REGION Network 6: Current revision and modification history
   // ▄▄▄▄▄▄▄▄▄▄▄▄▄▄▄▄▄▄▄▄▄▄▄▄▄▄▄▄▄▄▄▄▄▄▄▄▄▄▄▄▄▄▄▄
   // MODIFICATION HISTORY
   // 
   // 
   // The revision data shown here, in the network comments, contains additional information 
   // reflecting the software development workflow under the version control system (VCS) employed 
   // to track all software changes.
   // 
   // The VCS in use is the Git Source Code Management system in conjunction with the GitHub online 
   // hosting system. The software in its entirety is available in the GitHub remote repository:
   // 
   //      https://github.com/practicalseries/PS2001-pal-software
   // 
   // The repository is public and can be freely copied (forked in GitHub terminology) and used 
   // under the MIT licence. 
   // 
   // The MIT licence is reproduced in full in the last network of this software module.
   // 
   // 
   //  ―――――――――――――――――――――――――――――――――――――――――――
   //  DATE       REVISION             MASTER BRANCH     DEV
   //          (nnn.amm)   COMMIT TAG    (Base ---> Merge)    BRANCH   Author
   //  ———————————————————————————————————————————
   //  2022.04.16    002.000   D0011      D0010 D0011  None    M. Gledhill
   //                        FC11001 — RELEASED FOR USE
   //                          Merge back to master branch
   // 
   //  2022.04.11    001.801   D0010A-000.801   D0010 N/A     D010A   M. Gledhill
   //                        Released for test (SCV)
   // 
   //  2022.04.06    001.101   D0010A-000.104   D0010 N/A     D010A   M. Gledhill
   //                        Comments updated and standardised
   // 
   //  2021.08.23    001.000   D0009      D0008 D0009  None    M. Gledhill
   //                        FC11001 — RELEASED FOR USE
   //                          Merge back to master branch
   // 
   //  2021.08.23    001.000   D0008A-001.000   D0008 N/A     D0008A   M. Gledhill
   //                        FC11001 — Post-test RELEASED FOR USE
   // 
   //  2021.08.17    000.801   D0008A-000.801   D0008 N/A     D0008A   M. Gledhill
   //                        FC11001 Released for SMT
   // 
   //  2021.08.10    000.103   D0008A-000.103   D0008 N/A     D0008A   M. Gledhill
   //                        FC11001 Initial development testing
   // 
   //  2021.07.21    000.102   D0008A-000.102   D0008 N/A     D0008A   M. Gledhill
   //                        FC11001 Incremental build
   // 
   //  2021.07.13    000.101   D0008A-000.101   D0008 N/A     D0008A   M. Gledhill
   //                        FC11001 Block created — Comments added
   //  ———————————————————————————————————————————
   //   Where: nnn  =  Major revision
   //         a  =  Type (1-7 Development, 8 Proving, 9 Qualification, 0 Release)
   //       mm  =  Minor revision (must be 00 if a = 0)
   //         Block properties version number should be set to nn.a (only one decimal place)
   // 
   // ▄▄▄▄▄▄▄▄▄▄▄▄▄▄▄▄▄▄▄▄▄▄▄▄▄▄▄▄▄▄▄▄▄▄▄▄▄▄▄▄▄▄▄▄
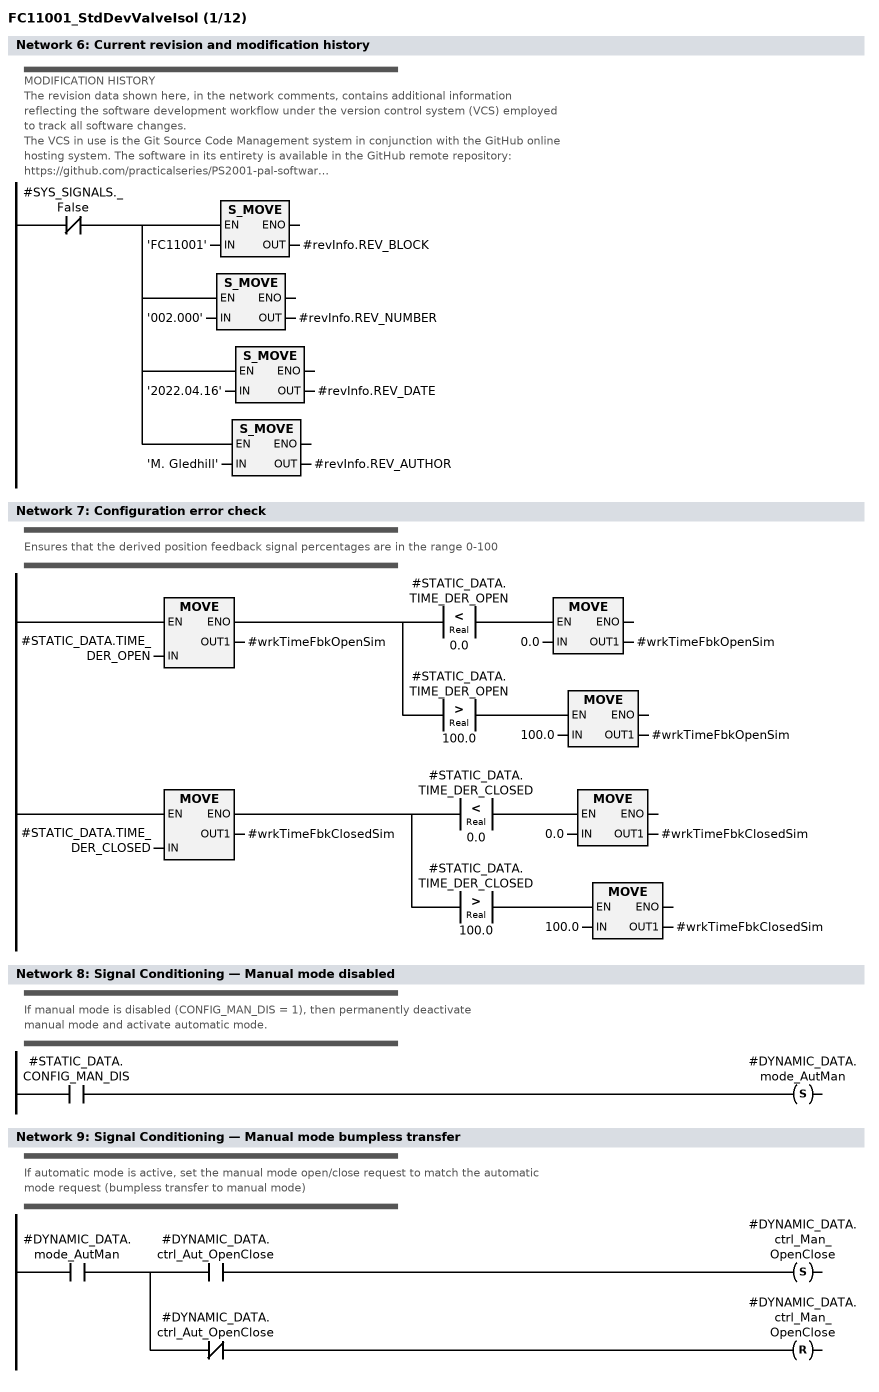
   RUNG wire#powerrail
      I_Contact( #SYS_SIGNALS._False )
      wire#w1
      S_Move(in := 'FC11001', out => #revInfo.REV_BLOCK)
   END_RUNG
   RUNG wire#w1
      S_Move(in := '002.000', out => #revInfo.REV_NUMBER)
   END_RUNG
   RUNG wire#w1
      S_Move(in := '2022.04.16', out => #revInfo.REV_DATE)
   END_RUNG
   RUNG wire#w1
      S_Move(in := 'M. Gledhill', out => #revInfo.REV_AUTHOR)
   END_RUNG
   // the same network as SCL:
   IF NOT #SYS_SIGNALS._False THEN
       #revInfo.REV_BLOCK := 'FC11001';
       #revInfo.REV_NUMBER := '002.000';
       #revInfo.REV_DATE := '2022.04.16';
       #revInfo.REV_AUTHOR := 'M. Gledhill';
   END_IF;
END_REGION

REGION Network 7: Configuration error check
   // ▀▀▀▀▀▀▀▀▀▀▀▀▀▀▀▀▀▀▀▀▀▀▀▀▀▀▀▀▀▀▀▀▀▀▀▀▀▀▀▀▀▀▀▀
   // Ensures that the derived position feedback signal percentages are in the range 0-100
   // ▄▄▄▄▄▄▄▄▄▄▄▄▄▄▄▄▄▄▄▄▄▄▄▄▄▄▄▄▄▄▄▄▄▄▄▄▄▄▄▄▄▄▄▄
   RUNG wire#powerrail
      Move(in := #STATIC_DATA.TIME_DER_OPEN, out1 => #wrkTimeFbkOpenSim)
      wire#w1
      { S7_Templates := "SrcType := Real" } LT_Contact(in1 := #STATIC_DATA.TIME_DER_OPEN, in2 := 0.0)
      Move(in := 0.0, out1 => #wrkTimeFbkOpenSim)
   END_RUNG
   RUNG wire#w1
      { S7_Templates := "SrcType := Real" } GT_Contact(in1 := #STATIC_DATA.TIME_DER_OPEN, in2 := 100.0)
      Move(in := 100.0, out1 => #wrkTimeFbkOpenSim)
   END_RUNG
   RUNG wire#powerrail
      Move(in := #STATIC_DATA.TIME_DER_CLOSED, out1 => #wrkTimeFbkClosedSim)
      wire#w2
      { S7_Templates := "SrcType := Real" } LT_Contact(in1 := #STATIC_DATA.TIME_DER_CLOSED, in2 := 0.0)
      Move(in := 0.0, out1 => #wrkTimeFbkClosedSim)
   END_RUNG
   RUNG wire#w2
      { S7_Templates := "SrcType := Real" } GT_Contact(in1 := #STATIC_DATA.TIME_DER_CLOSED, in2 := 100.0)
      Move(in := 100.0, out1 => #wrkTimeFbkClosedSim)
   END_RUNG
   // the same network as SCL:
   #wrkTimeFbkOpenSim := #STATIC_DATA.TIME_DER_OPEN;
   IF #STATIC_DATA.TIME_DER_OPEN < 0.0 THEN #wrkTimeFbkOpenSim := 0.0; END_IF;
   IF #STATIC_DATA.TIME_DER_OPEN > 100.0 THEN #wrkTimeFbkOpenSim := 100.0; END_IF;
   #wrkTimeFbkClosedSim := #STATIC_DATA.TIME_DER_CLOSED;
   IF #STATIC_DATA.TIME_DER_CLOSED < 0.0 THEN #wrkTimeFbkClosedSim := 0.0; END_IF;
   IF #STATIC_DATA.TIME_DER_CLOSED > 100.0 THEN #wrkTimeFbkClosedSim := 100.0; END_IF;
END_REGION

REGION Network 8: Signal Conditioning — Manual mode disabled
   // ▀▀▀▀▀▀▀▀▀▀▀▀▀▀▀▀▀▀▀▀▀▀▀▀▀▀▀▀▀▀▀▀▀▀▀▀▀▀▀▀▀▀▀▀
   // If manual mode is disabled (CONFIG_MAN_DIS = 1), then permanently deactivate
   // manual mode and activate automatic mode.
   // ▄▄▄▄▄▄▄▄▄▄▄▄▄▄▄▄▄▄▄▄▄▄▄▄▄▄▄▄▄▄▄▄▄▄▄▄▄▄▄▄▄▄▄▄
   RUNG wire#powerrail
      Contact( #STATIC_DATA.CONFIG_MAN_DIS )
      S_Coil( #DYNAMIC_DATA.mode_AutMan )
   END_RUNG
   // the same network as SCL:
   IF #STATIC_DATA.CONFIG_MAN_DIS THEN #DYNAMIC_DATA.mode_AutMan := TRUE; END_IF;
END_REGION

REGION Network 9: Signal Conditioning — Manual mode bumpless transfer
   // ▀▀▀▀▀▀▀▀▀▀▀▀▀▀▀▀▀▀▀▀▀▀▀▀▀▀▀▀▀▀▀▀▀▀▀▀▀▀▀▀▀▀▀▀
   // If automatic mode is active, set the manual mode open/close request to match the automatic
   // mode request (bumpless transfer to manual mode)
   // ▄▄▄▄▄▄▄▄▄▄▄▄▄▄▄▄▄▄▄▄▄▄▄▄▄▄▄▄▄▄▄▄▄▄▄▄▄▄▄▄▄▄▄▄
   RUNG wire#powerrail
      Contact( #DYNAMIC_DATA.mode_AutMan )
      wire#w1
      Contact( #DYNAMIC_DATA.ctrl_Aut_OpenClose )
      S_Coil( #DYNAMIC_DATA.ctrl_Man_OpenClose )
   END_RUNG
   RUNG wire#w1
      I_Contact( #DYNAMIC_DATA.ctrl_Aut_OpenClose )
      R_Coil( #DYNAMIC_DATA.ctrl_Man_OpenClose )
   END_RUNG
   // the same network as SCL:
   IF #DYNAMIC_DATA.mode_AutMan AND #DYNAMIC_DATA.ctrl_Aut_OpenClose THEN
       #DYNAMIC_DATA.ctrl_Man_OpenClose := TRUE;
   END_IF;
   IF #DYNAMIC_DATA.mode_AutMan AND NOT #DYNAMIC_DATA.ctrl_Aut_OpenClose THEN
       #DYNAMIC_DATA.ctrl_Man_OpenClose := FALSE;
   END_IF;
END_REGION

REGION Network 10: Signal Conditioning — Bypass mode disabled
   // ▀▀▀▀▀▀▀▀▀▀▀▀▀▀▀▀▀▀▀▀▀▀▀▀▀▀▀▀▀▀▀▀▀▀▀▀▀▀▀▀▀▀▀▀
   // If bypass mode is disabled (CONFIG_BYPASS_DIS = 1), then permanently deactivate
   // bypass mode.
   // ▄▄▄▄▄▄▄▄▄▄▄▄▄▄▄▄▄▄▄▄▄▄▄▄▄▄▄▄▄▄▄▄▄▄▄▄▄▄▄▄▄▄▄▄
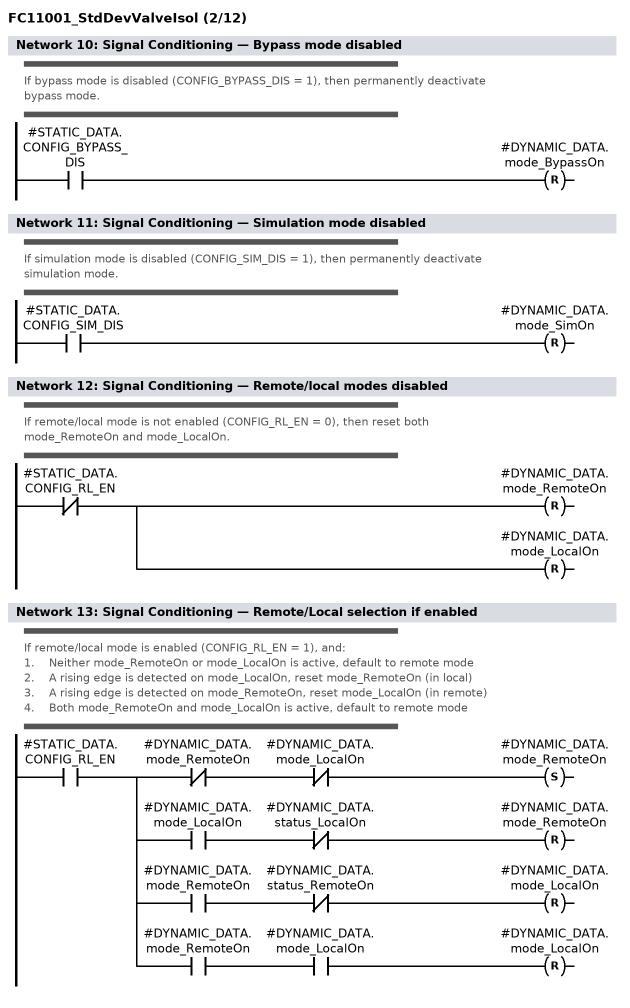
   RUNG wire#powerrail
      Contact( #STATIC_DATA.CONFIG_BYPASS_DIS )
      R_Coil( #DYNAMIC_DATA.mode_BypassOn )
   END_RUNG
   // the same network as SCL:
   IF #STATIC_DATA.CONFIG_BYPASS_DIS THEN #DYNAMIC_DATA.mode_BypassOn := FALSE; END_IF;
END_REGION

REGION Network 11: Signal Conditioning — Simulation mode disabled
   // ▀▀▀▀▀▀▀▀▀▀▀▀▀▀▀▀▀▀▀▀▀▀▀▀▀▀▀▀▀▀▀▀▀▀▀▀▀▀▀▀▀▀▀▀
   // If simulation mode is disabled (CONFIG_SIM_DIS = 1), then permanently deactivate
   // simulation mode.
   // ▄▄▄▄▄▄▄▄▄▄▄▄▄▄▄▄▄▄▄▄▄▄▄▄▄▄▄▄▄▄▄▄▄▄▄▄▄▄▄▄▄▄▄▄
   RUNG wire#powerrail
      Contact( #STATIC_DATA.CONFIG_SIM_DIS )
      R_Coil( #DYNAMIC_DATA.mode_SimOn )
   END_RUNG
   // the same network as SCL:
   IF #STATIC_DATA.CONFIG_SIM_DIS THEN #DYNAMIC_DATA.mode_SimOn := FALSE; END_IF;
END_REGION

REGION Network 12: Signal Conditioning — Remote/local modes disabled
   // ▀▀▀▀▀▀▀▀▀▀▀▀▀▀▀▀▀▀▀▀▀▀▀▀▀▀▀▀▀▀▀▀▀▀▀▀▀▀▀▀▀▀▀▀
   // If remote/local mode is not enabled (CONFIG_RL_EN = 0), then reset both 
   // mode_RemoteOn and mode_LocalOn.
   // ▄▄▄▄▄▄▄▄▄▄▄▄▄▄▄▄▄▄▄▄▄▄▄▄▄▄▄▄▄▄▄▄▄▄▄▄▄▄▄▄▄▄▄▄
   RUNG wire#powerrail
      I_Contact( #STATIC_DATA.CONFIG_RL_EN )
      wire#w1
      R_Coil( #DYNAMIC_DATA.mode_RemoteOn )
   END_RUNG
   RUNG wire#w1
      R_Coil( #DYNAMIC_DATA.mode_LocalOn )
   END_RUNG
   // the same network as SCL:
   IF NOT #STATIC_DATA.CONFIG_RL_EN THEN
       #DYNAMIC_DATA.mode_RemoteOn := FALSE;
       #DYNAMIC_DATA.mode_LocalOn := FALSE;
   END_IF;
END_REGION

REGION Network 13: Signal Conditioning — Remote/Local selection if enabled
   // ▀▀▀▀▀▀▀▀▀▀▀▀▀▀▀▀▀▀▀▀▀▀▀▀▀▀▀▀▀▀▀▀▀▀▀▀▀▀▀▀▀▀▀▀
   // If remote/local mode is enabled (CONFIG_RL_EN = 1), and:
   // 
   //    1.  Neither mode_RemoteOn or mode_LocalOn is active, default to remote mode
   //    2.  A rising edge is detected on mode_LocalOn, reset mode_RemoteOn (in local)
   //    3.  A rising edge is detected on mode_RemoteOn, reset mode_LocalOn (in remote)
   //    4.  Both mode_RemoteOn and mode_LocalOn is active, default to remote mode
   // ▄▄▄▄▄▄▄▄▄▄▄▄▄▄▄▄▄▄▄▄▄▄▄▄▄▄▄▄▄▄▄▄▄▄▄▄▄▄▄▄▄▄▄▄
   RUNG wire#powerrail
      Contact( #STATIC_DATA.CONFIG_RL_EN )
      wire#w1
      I_Contact( #DYNAMIC_DATA.mode_RemoteOn )
      I_Contact( #DYNAMIC_DATA.mode_LocalOn )
      S_Coil( #DYNAMIC_DATA.mode_RemoteOn )
   END_RUNG
   RUNG wire#w1
      Contact( #DYNAMIC_DATA.mode_LocalOn )
      I_Contact( #DYNAMIC_DATA.status_LocalOn )
      R_Coil( #DYNAMIC_DATA.mode_RemoteOn )
   END_RUNG
   RUNG wire#w1
      Contact( #DYNAMIC_DATA.mode_RemoteOn )
      I_Contact( #DYNAMIC_DATA.status_RemoteOn )
      R_Coil( #DYNAMIC_DATA.mode_LocalOn )
   END_RUNG
   RUNG wire#w1
      Contact( #DYNAMIC_DATA.mode_RemoteOn )
      Contact( #DYNAMIC_DATA.mode_LocalOn )
      R_Coil( #DYNAMIC_DATA.mode_LocalOn )
   END_RUNG
   // the same network as SCL:
   IF #STATIC_DATA.CONFIG_RL_EN AND NOT #DYNAMIC_DATA.mode_RemoteOn AND NOT #DYNAMIC_DATA.mode_LocalOn THEN
       #DYNAMIC_DATA.mode_RemoteOn := TRUE;
   END_IF;
   IF #STATIC_DATA.CONFIG_RL_EN AND #DYNAMIC_DATA.mode_LocalOn AND NOT #DYNAMIC_DATA.status_LocalOn THEN
       #DYNAMIC_DATA.mode_RemoteOn := FALSE;
   END_IF;
   IF #STATIC_DATA.CONFIG_RL_EN AND #DYNAMIC_DATA.mode_RemoteOn AND NOT #DYNAMIC_DATA.status_RemoteOn THEN
       #DYNAMIC_DATA.mode_LocalOn := FALSE;
   END_IF;
   IF #STATIC_DATA.CONFIG_RL_EN AND #DYNAMIC_DATA.mode_RemoteOn AND #DYNAMIC_DATA.mode_LocalOn THEN
       #DYNAMIC_DATA.mode_LocalOn := FALSE;
   END_IF;
END_REGION

REGION Network 14: Signal Conditioning — Derived open position
   // ▀▀▀▀▀▀▀▀▀▀▀▀▀▀▀▀▀▀▀▀▀▀▀▀▀▀▀▀▀▀▀▀▀▀▀▀▀▀▀▀▀▀▀▀
   // If there is no open position feedback (CONFIG_FBK_OPEN_EN = 0), then the open state of the 
   // valve is derived from the elapsed time of the operation timer using the following formulae:
   // 
   // ┌───────────────────────────────────────────┐
   // │$derived_fbk_open =1 when:                                │
   // │                                 wrkTimeFbkOpenSim  │
   // │actual_Operating_Timer ≤ TIME_OPENING_MAX ─ TIME_OPENING_MAX ╳ ----------------------------------------│
   // │                                     100     │
   // └───────────────────────────────────────────┘
   // Note:    wrkTimeFbkOpenSim is the error checked equivalent of TIME_FBK_OPEN
   // 
   // If the calculated elapsed time is close to or less than k_TIME_OP_MIN (210ms),
   // the calculated elapsed time (calOpenElapsedTime) is set to k_TIME_OP_MIN. This ensures at
   // least one timing pulse is required before the timer reaches zero.
   // 
   // The derived open signal ($derived_fbk_open) is reset if the valve is requested to be closed
   // ($ctrl_OpenClose = 0).
   // ▄▄▄▄▄▄▄▄▄▄▄▄▄▄▄▄▄▄▄▄▄▄▄▄▄▄▄▄▄▄▄▄▄▄▄▄▄▄▄▄▄▄▄▄
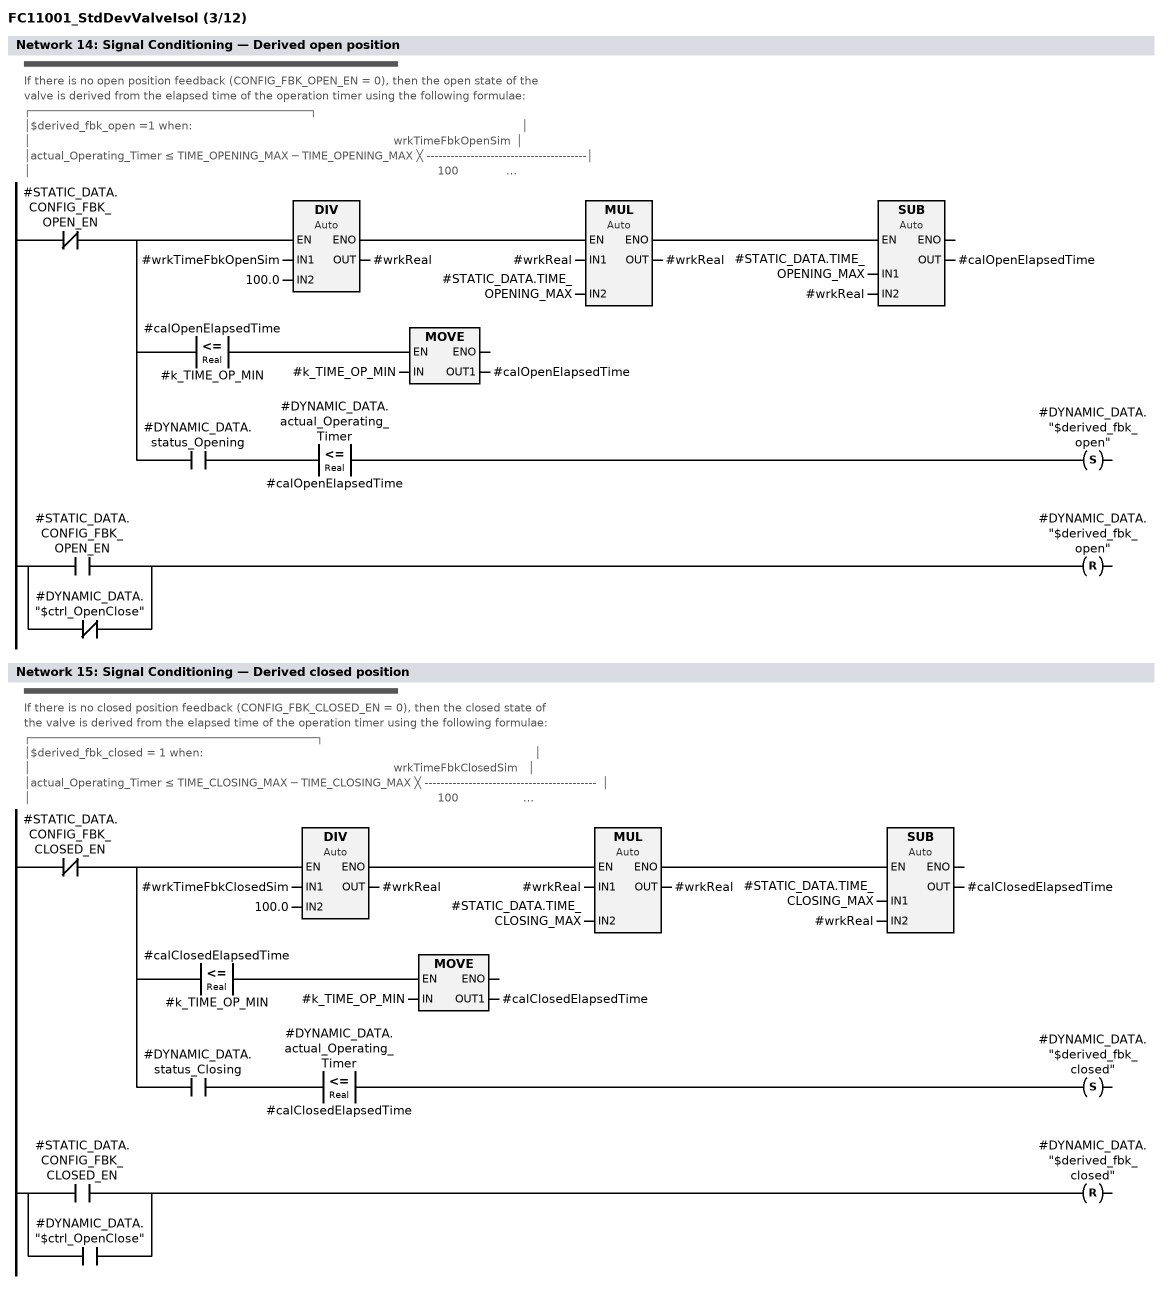
   RUNG wire#powerrail
      I_Contact( #STATIC_DATA.CONFIG_FBK_OPEN_EN )
      wire#w1
      Div(in1 := #wrkTimeFbkOpenSim, in2 := 100.0, out => #wrkReal)
      Mul(in1 := #wrkReal, in2 := #STATIC_DATA.TIME_OPENING_MAX, out => #wrkReal)
      Sub(in1 := #STATIC_DATA.TIME_OPENING_MAX, in2 := #wrkReal, out => #calOpenElapsedTime)
   END_RUNG
   RUNG wire#w1
      { S7_Templates := "SrcType := Real" } LE_Contact(in1 := #calOpenElapsedTime, in2 := #k_TIME_OP_MIN)
      Move(in := #k_TIME_OP_MIN, out1 => #calOpenElapsedTime)
   END_RUNG
   RUNG wire#w1
      Contact( #DYNAMIC_DATA.status_Opening )
      { S7_Templates := "SrcType := Real" } LE_Contact(in1 := #DYNAMIC_DATA.actual_Operating_Timer, in2 := #calOpenElapsedTime)
      S_Coil( #DYNAMIC_DATA."$derived_fbk_open" )
   END_RUNG
   RUNG wire#powerrail
      Contact( #STATIC_DATA.CONFIG_FBK_OPEN_EN )
      wire#w2
      R_Coil( #DYNAMIC_DATA."$derived_fbk_open" )
   END_RUNG
   RUNG wire#powerrail
      I_Contact( #DYNAMIC_DATA."$ctrl_OpenClose" )
   END_RUNG wire#w2
   // the same network as SCL:
   #_w1 := NOT #STATIC_DATA.CONFIG_FBK_OPEN_EN;
   IF #_w1 THEN
       #wrkReal := #wrkTimeFbkOpenSim / 100.0;
       #wrkReal := #wrkReal * #STATIC_DATA.TIME_OPENING_MAX;
       #calOpenElapsedTime := #STATIC_DATA.TIME_OPENING_MAX - #wrkReal;
   END_IF;
   IF #_w1 AND (#calOpenElapsedTime <= #k_TIME_OP_MIN) THEN #calOpenElapsedTime := #k_TIME_OP_MIN; END_IF;
   IF #_w1 AND #DYNAMIC_DATA.status_Opening AND (#DYNAMIC_DATA.actual_Operating_Timer <= #calOpenElapsedTime) THEN
       #DYNAMIC_DATA."$derived_fbk_open" := TRUE;
   END_IF;
   IF #STATIC_DATA.CONFIG_FBK_OPEN_EN OR NOT #DYNAMIC_DATA."$ctrl_OpenClose" THEN
       #DYNAMIC_DATA."$derived_fbk_open" := FALSE;
   END_IF;
END_REGION

REGION Network 15: Signal Conditioning — Derived closed position
   // ▀▀▀▀▀▀▀▀▀▀▀▀▀▀▀▀▀▀▀▀▀▀▀▀▀▀▀▀▀▀▀▀▀▀▀▀▀▀▀▀▀▀▀▀
   // If there is no closed position feedback (CONFIG_FBK_CLOSED_EN = 0), then the closed state of 
   // the valve is derived from the elapsed time of the operation timer using the following formulae:
   // 
   // ┌────────────────────────────────────────────┐
   // │$derived_fbk_closed = 1 when:                                 │
   // │                                 wrkTimeFbkClosedSim   │
   // │actual_Operating_Timer ≤ TIME_CLOSING_MAX ─ TIME_CLOSING_MAX ╳ -------------------------------------------  │
   // │                                     100            │
   // └────────────────────────────────────────────┘
   // Note:    wrkTimeFbkClosedSim is the error checked equivalent of TIME_FBK_CLOSED
   // 
   // If the calculated elapsed time is close to or less than k_TIME_OP_MIN (210ms),
   // the calculated elapsed time (calClosedElapsedTime) is set to k_TIME_OP_MIN. This ensures at
   // least one timing pulse is required before the timer reaches zero.
   // 
   // The derived closed signal ($derived_fbk_closed) is reset if the valve is requested to be open
   // ($ctrl_OpenClose = 1).
   // ▄▄▄▄▄▄▄▄▄▄▄▄▄▄▄▄▄▄▄▄▄▄▄▄▄▄▄▄▄▄▄▄▄▄▄▄▄▄▄▄▄▄▄▄
   RUNG wire#powerrail
      I_Contact( #STATIC_DATA.CONFIG_FBK_CLOSED_EN )
      wire#w1
      Div(in1 := #wrkTimeFbkClosedSim, in2 := 100.0, out => #wrkReal)
      Mul(in1 := #wrkReal, in2 := #STATIC_DATA.TIME_CLOSING_MAX, out => #wrkReal)
      Sub(in1 := #STATIC_DATA.TIME_CLOSING_MAX, in2 := #wrkReal, out => #calClosedElapsedTime)
   END_RUNG
   RUNG wire#w1
      { S7_Templates := "SrcType := Real" } LE_Contact(in1 := #calClosedElapsedTime, in2 := #k_TIME_OP_MIN)
      Move(in := #k_TIME_OP_MIN, out1 => #calClosedElapsedTime)
   END_RUNG
   RUNG wire#w1
      Contact( #DYNAMIC_DATA.status_Closing )
      { S7_Templates := "SrcType := Real" } LE_Contact(in1 := #DYNAMIC_DATA.actual_Operating_Timer, in2 := #calClosedElapsedTime)
      S_Coil( #DYNAMIC_DATA."$derived_fbk_closed" )
   END_RUNG
   RUNG wire#powerrail
      Contact( #STATIC_DATA.CONFIG_FBK_CLOSED_EN )
      wire#w2
      R_Coil( #DYNAMIC_DATA."$derived_fbk_closed" )
   END_RUNG
   RUNG wire#powerrail
      Contact( #DYNAMIC_DATA."$ctrl_OpenClose" )
   END_RUNG wire#w2
   // the same network as SCL:
   #_w1 := NOT #STATIC_DATA.CONFIG_FBK_CLOSED_EN;
   IF #_w1 THEN
       #wrkReal := #wrkTimeFbkClosedSim / 100.0;
       #wrkReal := #wrkReal * #STATIC_DATA.TIME_CLOSING_MAX;
       #calClosedElapsedTime := #STATIC_DATA.TIME_CLOSING_MAX - #wrkReal;
   END_IF;
   IF #_w1 AND (#calClosedElapsedTime <= #k_TIME_OP_MIN) THEN
       #calClosedElapsedTime := #k_TIME_OP_MIN;
   END_IF;
   IF #_w1 AND #DYNAMIC_DATA.status_Closing AND (#DYNAMIC_DATA.actual_Operating_Timer <= #calClosedElapsedTime) THEN
       #DYNAMIC_DATA."$derived_fbk_closed" := TRUE;
   END_IF;
   IF #STATIC_DATA.CONFIG_FBK_CLOSED_EN OR #DYNAMIC_DATA."$ctrl_OpenClose" THEN
       #DYNAMIC_DATA."$derived_fbk_closed" := FALSE;
   END_IF;
END_REGION

REGION Network 16: Signal Conditioning — Simulation mode — Open signal
   // ▀▀▀▀▀▀▀▀▀▀▀▀▀▀▀▀▀▀▀▀▀▀▀▀▀▀▀▀▀▀▀▀▀▀▀▀▀▀▀▀▀▀▀▀
   // If simulation mode is active, the simulated open position signal is set as follows:
   // 
   //    •   mode_SimValue = 0 (no feedback), $sim_fbk_open = 0
   // 
   //    •   mode_SimValue = 1 (permanently open), $sim_fbk_open = 1
   // 
   //    •   mode_SimValue = 2 (permanently closed), $sim_fbk_open = 0
   // 
   //    •   mode_SimValue = 3 (follow demand), $sim_fbk_open = $ctrl_OpenClose
   // 
   // If simulation mode is not active,  $sim_fbk_open = 0
   // ▄▄▄▄▄▄▄▄▄▄▄▄▄▄▄▄▄▄▄▄▄▄▄▄▄▄▄▄▄▄▄▄▄▄▄▄▄▄▄▄▄▄▄▄
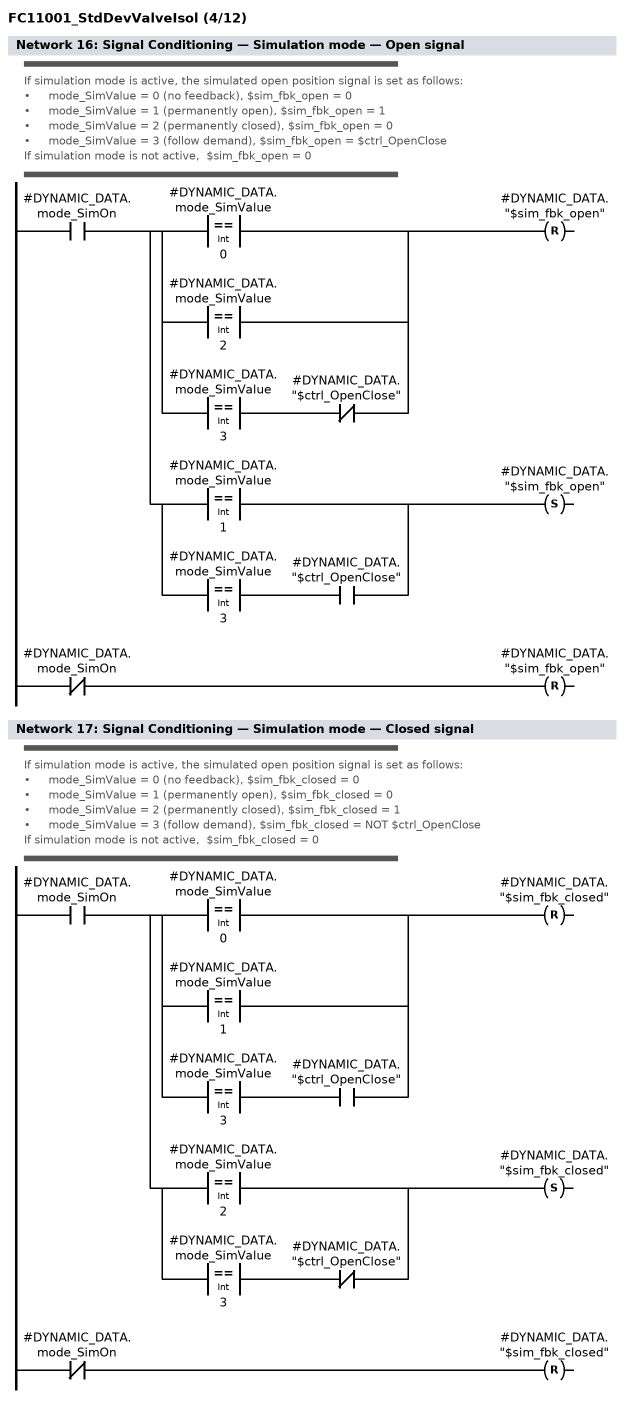
   RUNG wire#powerrail
      Contact( #DYNAMIC_DATA.mode_SimOn )
      wire#w1
      { S7_Templates := "SrcType := Int" } EQ_Contact(in1 := #DYNAMIC_DATA.mode_SimValue, in2 := 0)
      wire#w2
      R_Coil( #DYNAMIC_DATA."$sim_fbk_open" )
   END_RUNG
   RUNG wire#w1
      { S7_Templates := "SrcType := Int" } EQ_Contact(in1 := #DYNAMIC_DATA.mode_SimValue, in2 := 2)
   END_RUNG wire#w2
   RUNG wire#w1
      { S7_Templates := "SrcType := Int" } EQ_Contact(in1 := #DYNAMIC_DATA.mode_SimValue, in2 := 3)
      I_Contact( #DYNAMIC_DATA."$ctrl_OpenClose" )
   END_RUNG wire#w2
   RUNG wire#w1
      { S7_Templates := "SrcType := Int" } EQ_Contact(in1 := #DYNAMIC_DATA.mode_SimValue, in2 := 1)
      wire#w3
      S_Coil( #DYNAMIC_DATA."$sim_fbk_open" )
   END_RUNG
   RUNG wire#w1
      { S7_Templates := "SrcType := Int" } EQ_Contact(in1 := #DYNAMIC_DATA.mode_SimValue, in2 := 3)
      Contact( #DYNAMIC_DATA."$ctrl_OpenClose" )
   END_RUNG wire#w3
   RUNG wire#powerrail
      I_Contact( #DYNAMIC_DATA.mode_SimOn )
      R_Coil( #DYNAMIC_DATA."$sim_fbk_open" )
   END_RUNG
   // the same network as SCL:
   IF #DYNAMIC_DATA.mode_SimOn AND ((#DYNAMIC_DATA.mode_SimValue = 0) OR (#DYNAMIC_DATA.mode_SimValue = 2) OR ((#DYNAMIC_DATA.mode_SimValue = 3) AND NOT #DYNAMIC_DATA."$ctrl_OpenClose")) THEN
       #DYNAMIC_DATA."$sim_fbk_open" := FALSE;
   END_IF;
   IF #DYNAMIC_DATA.mode_SimOn AND ((#DYNAMIC_DATA.mode_SimValue = 1) OR ((#DYNAMIC_DATA.mode_SimValue = 3) AND #DYNAMIC_DATA."$ctrl_OpenClose")) THEN
       #DYNAMIC_DATA."$sim_fbk_open" := TRUE;
   END_IF;
   IF NOT #DYNAMIC_DATA.mode_SimOn THEN #DYNAMIC_DATA."$sim_fbk_open" := FALSE; END_IF;
END_REGION

REGION Network 17: Signal Conditioning — Simulation mode — Closed signal
   // ▀▀▀▀▀▀▀▀▀▀▀▀▀▀▀▀▀▀▀▀▀▀▀▀▀▀▀▀▀▀▀▀▀▀▀▀▀▀▀▀▀▀▀▀
   // If simulation mode is active, the simulated open position signal is set as follows:
   // 
   //    •   mode_SimValue = 0 (no feedback), $sim_fbk_closed = 0
   // 
   //    •   mode_SimValue = 1 (permanently open), $sim_fbk_closed = 0
   // 
   //    •   mode_SimValue = 2 (permanently closed), $sim_fbk_closed = 1
   // 
   //    •   mode_SimValue = 3 (follow demand), $sim_fbk_closed = NOT $ctrl_OpenClose
   // 
   // If simulation mode is not active,  $sim_fbk_closed = 0
   // ▄▄▄▄▄▄▄▄▄▄▄▄▄▄▄▄▄▄▄▄▄▄▄▄▄▄▄▄▄▄▄▄▄▄▄▄▄▄▄▄▄▄▄▄
   RUNG wire#powerrail
      Contact( #DYNAMIC_DATA.mode_SimOn )
      wire#w1
      { S7_Templates := "SrcType := Int" } EQ_Contact(in1 := #DYNAMIC_DATA.mode_SimValue, in2 := 0)
      wire#w2
      R_Coil( #DYNAMIC_DATA."$sim_fbk_closed" )
   END_RUNG
   RUNG wire#w1
      { S7_Templates := "SrcType := Int" } EQ_Contact(in1 := #DYNAMIC_DATA.mode_SimValue, in2 := 1)
   END_RUNG wire#w2
   RUNG wire#w1
      { S7_Templates := "SrcType := Int" } EQ_Contact(in1 := #DYNAMIC_DATA.mode_SimValue, in2 := 3)
      Contact( #DYNAMIC_DATA."$ctrl_OpenClose" )
   END_RUNG wire#w2
   RUNG wire#w1
      { S7_Templates := "SrcType := Int" } EQ_Contact(in1 := #DYNAMIC_DATA.mode_SimValue, in2 := 2)
      wire#w3
      S_Coil( #DYNAMIC_DATA."$sim_fbk_closed" )
   END_RUNG
   RUNG wire#w1
      { S7_Templates := "SrcType := Int" } EQ_Contact(in1 := #DYNAMIC_DATA.mode_SimValue, in2 := 3)
      I_Contact( #DYNAMIC_DATA."$ctrl_OpenClose" )
   END_RUNG wire#w3
   RUNG wire#powerrail
      I_Contact( #DYNAMIC_DATA.mode_SimOn )
      R_Coil( #DYNAMIC_DATA."$sim_fbk_closed" )
   END_RUNG
   // the same network as SCL:
   IF #DYNAMIC_DATA.mode_SimOn AND ((#DYNAMIC_DATA.mode_SimValue = 0) OR (#DYNAMIC_DATA.mode_SimValue = 1) OR ((#DYNAMIC_DATA.mode_SimValue = 3) AND #DYNAMIC_DATA."$ctrl_OpenClose")) THEN
       #DYNAMIC_DATA."$sim_fbk_closed" := FALSE;
   END_IF;
   IF #DYNAMIC_DATA.mode_SimOn AND ((#DYNAMIC_DATA.mode_SimValue = 2) OR ((#DYNAMIC_DATA.mode_SimValue = 3) AND NOT #DYNAMIC_DATA."$ctrl_OpenClose")) THEN
       #DYNAMIC_DATA."$sim_fbk_closed" := TRUE;
   END_IF;
   IF NOT #DYNAMIC_DATA.mode_SimOn THEN #DYNAMIC_DATA."$sim_fbk_closed" := FALSE; END_IF;
END_REGION

REGION Network 18: Signal conditioning — Determine valve OPEN position status
   // ▀▀▀▀▀▀▀▀▀▀▀▀▀▀▀▀▀▀▀▀▀▀▀▀▀▀▀▀▀▀▀▀▀▀▀▀▀▀▀▀▀▀▀▀
   // Generates a working open signal (wrkOpen), that is then used throughout the module as the 
   // definitive open position feedback signal.
   // 
   // The open signal will be either :
   // 
   //    1.  The same as the FBK_OPEN parameter if this is in use 
   //      (CONFIG_FBK_OPEN_EN = 1)
   // 
   //    2.  The internally derived open state (based on the requested state of the valve) if the 
   //      FBK_OPEN signal is NOT in use (CONFIG_FBK_OPEN_EN = 0)
   // 
   //    3.  The simulated state of the valve if simulation mode is active (mode_SimOn = 1)
   // 
   // If an actual open position signal is provided to the module via the FBK_OPEN parameter 
   // (i.e. if CONFIG_FBK_OPEN_EN = 1) then wrkOpen is set to match the FBK_OPEN signal 
   // (wrkOpen = FBK_OPEN).
   // 
   // If a derived open signal is to be used (i.e. if CONFIG_FBK_OPEN_EN = 0), then wrkOpen is set to 
   // match the internally derived $derived_fbk_open signal (wrkOpen = $derived_fbk_open). 
   // $derived_fbk_open is based on the requested state of the valve. 
   // 
   // Finally, if simulation mode is active (mode_SimOn = 1), then wrkOpen is set to match the internal 
   // simulation signal $sim_fbk_open signal (wrkOpen = $sim_fbk_open).. 
   // ▄▄▄▄▄▄▄▄▄▄▄▄▄▄▄▄▄▄▄▄▄▄▄▄▄▄▄▄▄▄▄▄▄▄▄▄▄▄▄▄▄▄▄▄
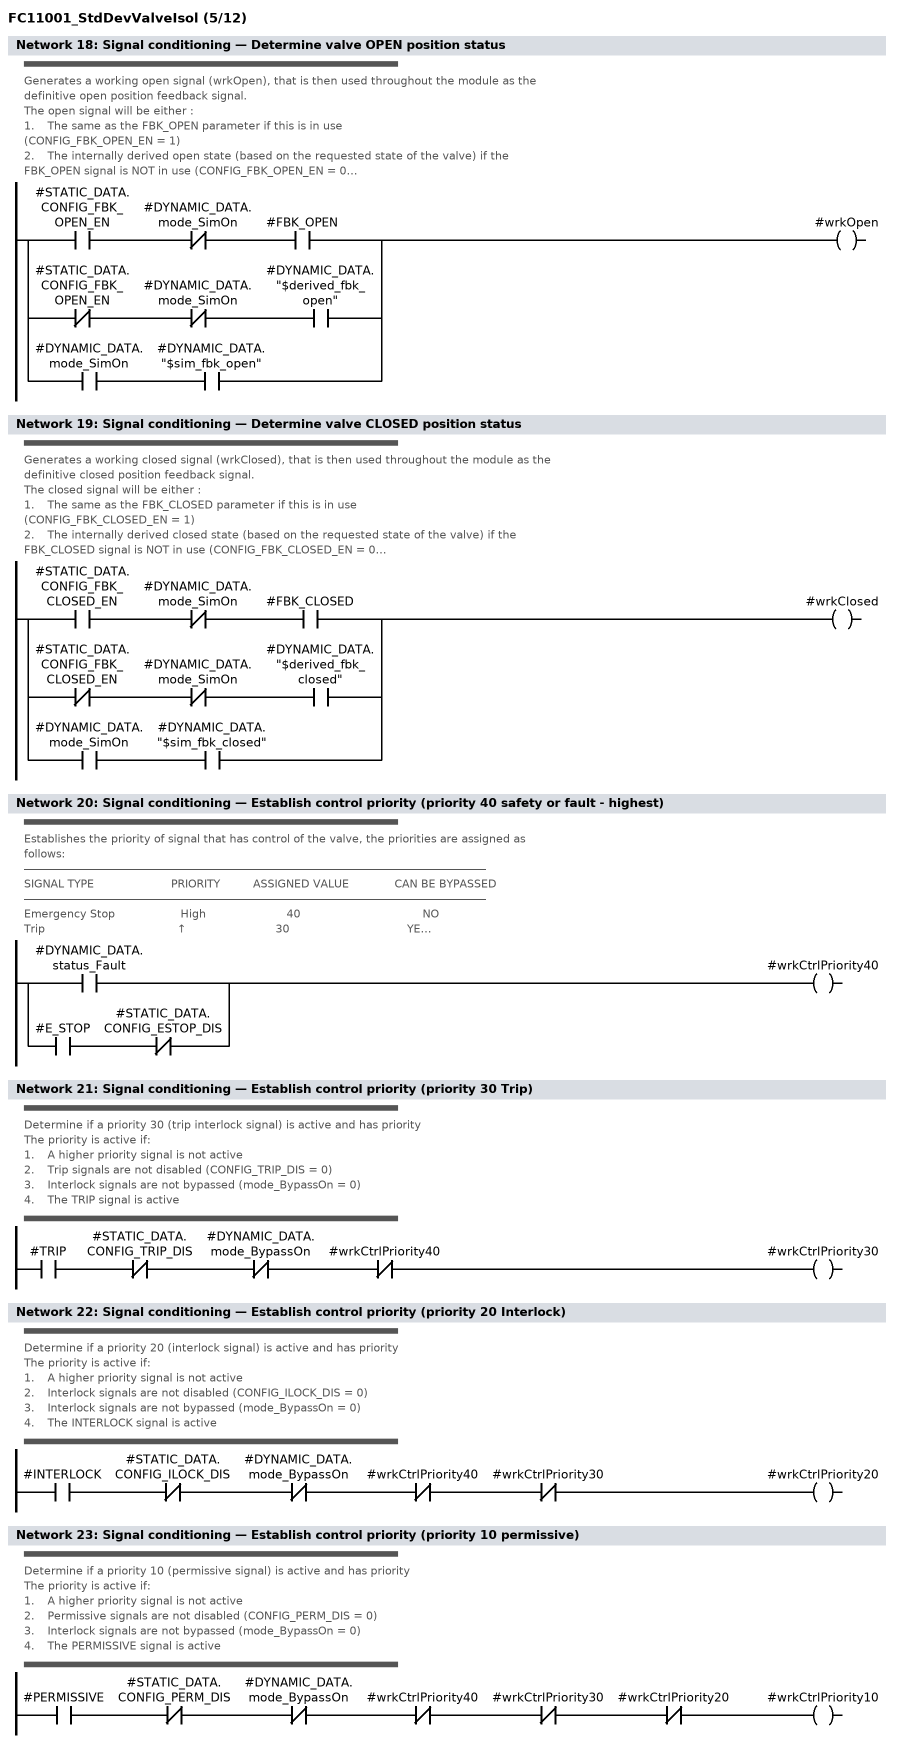
   RUNG wire#powerrail
      Contact( #STATIC_DATA.CONFIG_FBK_OPEN_EN )
      I_Contact( #DYNAMIC_DATA.mode_SimOn )
      Contact( #FBK_OPEN )
      wire#w1
      Coil( #wrkOpen )
   END_RUNG
   RUNG wire#powerrail
      I_Contact( #STATIC_DATA.CONFIG_FBK_OPEN_EN )
      I_Contact( #DYNAMIC_DATA.mode_SimOn )
      Contact( #DYNAMIC_DATA."$derived_fbk_open" )
   END_RUNG wire#w1
   RUNG wire#powerrail
      Contact( #DYNAMIC_DATA.mode_SimOn )
      Contact( #DYNAMIC_DATA."$sim_fbk_open" )
   END_RUNG wire#w1
   // the same network as SCL:
   #wrkOpen := (#STATIC_DATA.CONFIG_FBK_OPEN_EN AND NOT #DYNAMIC_DATA.mode_SimOn AND #FBK_OPEN) OR (NOT #STATIC_DATA.CONFIG_FBK_OPEN_EN AND NOT #DYNAMIC_DATA.mode_SimOn AND #DYNAMIC_DATA."$derived_fbk_open") OR (#DYNAMIC_DATA.mode_SimOn AND #DYNAMIC_DATA."$sim_fbk_open");
END_REGION

REGION Network 19: Signal conditioning — Determine valve CLOSED position status
   // ▀▀▀▀▀▀▀▀▀▀▀▀▀▀▀▀▀▀▀▀▀▀▀▀▀▀▀▀▀▀▀▀▀▀▀▀▀▀▀▀▀▀▀▀
   // Generates a working closed signal (wrkClosed), that is then used throughout the module as the 
   // definitive closed position feedback signal.
   // 
   // The closed signal will be either :
   // 
   //    1.  The same as the FBK_CLOSED parameter if this is in use 
   //      (CONFIG_FBK_CLOSED_EN = 1)
   // 
   //    2.  The internally derived closed state (based on the requested state of the valve) if the 
   //      FBK_CLOSED signal is NOT in use (CONFIG_FBK_CLOSED_EN = 0)
   // 
   //    3.  The simulated state of the valve if simulation mode is active (mode_SimOn = 1)
   // 
   // If an actual closed position signal is provided to the module via the FBK_CLOSED parameter 
   // (i.e. if CONFIG_FBK_CLOSED_EN = 1) then wrkClosed is set to match the FBK_CLOSED signal 
   // wrkClosed = FBK_CLOSED).
   // 
   // If a derived closed signal is to be used (i.e. if CONFIG_FBK_CLOSED_EN = 0), then wrkClosed is 
   // set to match the internally derived $derived_fbk_closed signal 
   // (wrkClosed = $derived_fbk_closed). $derived_fbk_closed is based on the requested state of 
   // the valve.
   // 
   // Finally, if simulation mode is active (mode_SimOn = 1), then wrkClosed is set to match the 
   // internal simulation signal $sim_fbk_closed signal (wrkClosed = $sim_fbk_closed). 
   // ▄▄▄▄▄▄▄▄▄▄▄▄▄▄▄▄▄▄▄▄▄▄▄▄▄▄▄▄▄▄▄▄▄▄▄▄▄▄▄▄▄▄▄▄
   RUNG wire#powerrail
      Contact( #STATIC_DATA.CONFIG_FBK_CLOSED_EN )
      I_Contact( #DYNAMIC_DATA.mode_SimOn )
      Contact( #FBK_CLOSED )
      wire#w1
      Coil( #wrkClosed )
   END_RUNG
   RUNG wire#powerrail
      I_Contact( #STATIC_DATA.CONFIG_FBK_CLOSED_EN )
      I_Contact( #DYNAMIC_DATA.mode_SimOn )
      Contact( #DYNAMIC_DATA."$derived_fbk_closed" )
   END_RUNG wire#w1
   RUNG wire#powerrail
      Contact( #DYNAMIC_DATA.mode_SimOn )
      Contact( #DYNAMIC_DATA."$sim_fbk_closed" )
   END_RUNG wire#w1
   // the same network as SCL:
   #wrkClosed := (#STATIC_DATA.CONFIG_FBK_CLOSED_EN AND NOT #DYNAMIC_DATA.mode_SimOn AND #FBK_CLOSED) OR (NOT #STATIC_DATA.CONFIG_FBK_CLOSED_EN AND NOT #DYNAMIC_DATA.mode_SimOn AND #DYNAMIC_DATA."$derived_fbk_closed") OR (#DYNAMIC_DATA.mode_SimOn AND #DYNAMIC_DATA."$sim_fbk_closed");
END_REGION

REGION Network 20: Signal conditioning — Establish control priority (priority 40 safety or fault - highest)
   // ▀▀▀▀▀▀▀▀▀▀▀▀▀▀▀▀▀▀▀▀▀▀▀▀▀▀▀▀▀▀▀▀▀▀▀▀▀▀▀▀▀▀▀▀
   // Establishes the priority of signal that has control of the valve, the priorities are assigned as 
   // follows:
   // 
   //  ――――――――――――――――――――――――――――――――――――――――――
   //  SIGNAL TYPE       PRIORITY   ASSIGNED VALUE       CAN BE BYPASSED
   //  ――――――――――――――――――――――――――――――――――――――――――
   //  Emergency Stop        High        40                NO
   //  Trip            ↑           30             YES
   //  Interlock            ↑           20             YES
   //  Permissive          ↑           10             YES
   //  Auto/manual control    Low         00                NO
   //  ――――――――――――――――――――――――――――――――――――――――――
   //  High priority signal take precedence over lower priority signals.
   // 
   // Determine a priority 40 (valve safety (or fault) condition is active)
   // 
   // The priority is active if:
   // 
   //    1.  The valve is in a fault condition (status_Fault = 1)
   // 
   //   OR both the following are true
   // 
   //    1.  Safety signals are not disabled (CONFIG_ESTOP_DIS = 0)
   // 
   //    2.  The E_STOP signal is active
   // ▄▄▄▄▄▄▄▄▄▄▄▄▄▄▄▄▄▄▄▄▄▄▄▄▄▄▄▄▄▄▄▄▄▄▄▄▄▄▄▄▄▄▄▄
   RUNG wire#powerrail
      Contact( #DYNAMIC_DATA.status_Fault )
      wire#w1
      Coil( #wrkCtrlPriority40 )
   END_RUNG
   RUNG wire#powerrail
      Contact( #E_STOP )
      I_Contact( #STATIC_DATA.CONFIG_ESTOP_DIS )
   END_RUNG wire#w1
   // the same network as SCL:
   #wrkCtrlPriority40 := #DYNAMIC_DATA.status_Fault OR (#E_STOP AND NOT #STATIC_DATA.CONFIG_ESTOP_DIS);
END_REGION

REGION Network 21: Signal conditioning — Establish control priority (priority 30 Trip)
   // ▀▀▀▀▀▀▀▀▀▀▀▀▀▀▀▀▀▀▀▀▀▀▀▀▀▀▀▀▀▀▀▀▀▀▀▀▀▀▀▀▀▀▀▀
   // Determine if a priority 30 (trip interlock signal) is active and has priority
   // 
   // The priority is active if:
   // 
   //    1.  A higher priority signal is not active
   // 
   //    2.  Trip signals are not disabled (CONFIG_TRIP_DIS = 0)
   // 
   //    3.  Interlock signals are not bypassed (mode_BypassOn = 0)
   // 
   //    4.  The TRIP signal is active
   // ▄▄▄▄▄▄▄▄▄▄▄▄▄▄▄▄▄▄▄▄▄▄▄▄▄▄▄▄▄▄▄▄▄▄▄▄▄▄▄▄▄▄▄▄
   RUNG wire#powerrail
      Contact( #TRIP )
      I_Contact( #STATIC_DATA.CONFIG_TRIP_DIS )
      I_Contact( #DYNAMIC_DATA.mode_BypassOn )
      I_Contact( #wrkCtrlPriority40 )
      Coil( #wrkCtrlPriority30 )
   END_RUNG
   // the same network as SCL:
   #wrkCtrlPriority30 := #TRIP AND NOT #STATIC_DATA.CONFIG_TRIP_DIS AND NOT #DYNAMIC_DATA.mode_BypassOn AND NOT #wrkCtrlPriority40;
END_REGION

REGION Network 22: Signal conditioning — Establish control priority (priority 20 Interlock)
   // ▀▀▀▀▀▀▀▀▀▀▀▀▀▀▀▀▀▀▀▀▀▀▀▀▀▀▀▀▀▀▀▀▀▀▀▀▀▀▀▀▀▀▀▀
   // Determine if a priority 20 (interlock signal) is active and has priority
   // 
   // The priority is active if:
   // 
   //    1.  A higher priority signal is not active
   // 
   //    2.  Interlock signals are not disabled (CONFIG_ILOCK_DIS = 0)
   // 
   //    3.  Interlock signals are not bypassed (mode_BypassOn = 0)
   // 
   //    4.  The INTERLOCK signal is active
   // ▄▄▄▄▄▄▄▄▄▄▄▄▄▄▄▄▄▄▄▄▄▄▄▄▄▄▄▄▄▄▄▄▄▄▄▄▄▄▄▄▄▄▄▄
   RUNG wire#powerrail
      Contact( #INTERLOCK )
      I_Contact( #STATIC_DATA.CONFIG_ILOCK_DIS )
      I_Contact( #DYNAMIC_DATA.mode_BypassOn )
      I_Contact( #wrkCtrlPriority40 )
      I_Contact( #wrkCtrlPriority30 )
      Coil( #wrkCtrlPriority20 )
   END_RUNG
   // the same network as SCL:
   #wrkCtrlPriority20 := #INTERLOCK AND NOT #STATIC_DATA.CONFIG_ILOCK_DIS AND NOT #DYNAMIC_DATA.mode_BypassOn AND NOT #wrkCtrlPriority40 AND NOT #wrkCtrlPriority30;
END_REGION

REGION Network 23: Signal conditioning — Establish control priority (priority 10 permissive)
   // ▀▀▀▀▀▀▀▀▀▀▀▀▀▀▀▀▀▀▀▀▀▀▀▀▀▀▀▀▀▀▀▀▀▀▀▀▀▀▀▀▀▀▀▀
   // Determine if a priority 10 (permissive signal) is active and has priority
   // 
   // The priority is active if:
   // 
   //    1.  A higher priority signal is not active
   // 
   //    2.  Permissive signals are not disabled (CONFIG_PERM_DIS = 0)
   // 
   //    3.  Interlock signals are not bypassed (mode_BypassOn = 0)
   // 
   //    4.  The PERMISSIVE signal is active
   // ▄▄▄▄▄▄▄▄▄▄▄▄▄▄▄▄▄▄▄▄▄▄▄▄▄▄▄▄▄▄▄▄▄▄▄▄▄▄▄▄▄▄▄▄
   RUNG wire#powerrail
      Contact( #PERMISSIVE )
      I_Contact( #STATIC_DATA.CONFIG_PERM_DIS )
      I_Contact( #DYNAMIC_DATA.mode_BypassOn )
      I_Contact( #wrkCtrlPriority40 )
      I_Contact( #wrkCtrlPriority30 )
      I_Contact( #wrkCtrlPriority20 )
      Coil( #wrkCtrlPriority10 )
   END_RUNG
   // the same network as SCL:
   #wrkCtrlPriority10 := #PERMISSIVE AND NOT #STATIC_DATA.CONFIG_PERM_DIS AND NOT #DYNAMIC_DATA.mode_BypassOn AND NOT #wrkCtrlPriority40 AND NOT #wrkCtrlPriority30 AND NOT #wrkCtrlPriority20;
END_REGION

REGION Network 24: Signal conditioning — Establish control priority (priority 00 auto/manual - lowest)
   // ▀▀▀▀▀▀▀▀▀▀▀▀▀▀▀▀▀▀▀▀▀▀▀▀▀▀▀▀▀▀▀▀▀▀▀▀▀▀▀▀▀▀▀▀
   // Determine if a priority 00 (automatic or manual control) is active and has priority
   // 
   // The priority is active if:
   // 
   //    1.  A higher priority signal is not active
   // ▄▄▄▄▄▄▄▄▄▄▄▄▄▄▄▄▄▄▄▄▄▄▄▄▄▄▄▄▄▄▄▄▄▄▄▄▄▄▄▄▄▄▄▄
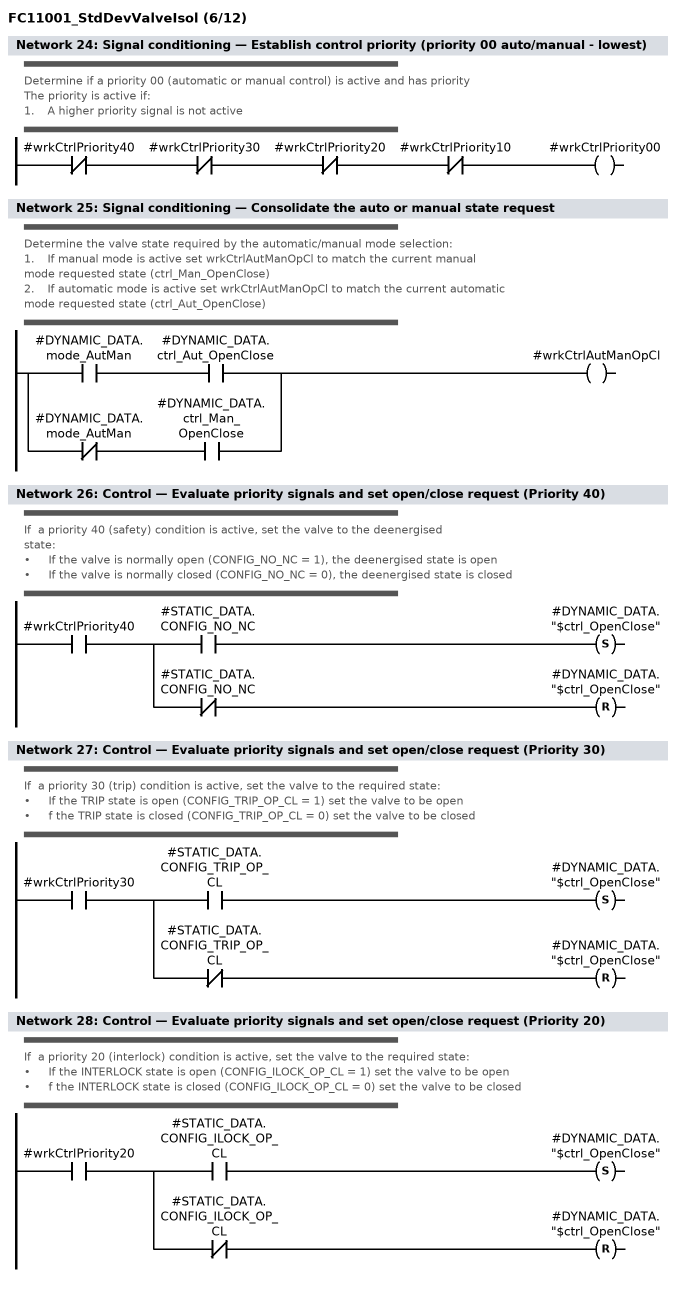
   RUNG wire#powerrail
      I_Contact( #wrkCtrlPriority40 )
      I_Contact( #wrkCtrlPriority30 )
      I_Contact( #wrkCtrlPriority20 )
      I_Contact( #wrkCtrlPriority10 )
      Coil( #wrkCtrlPriority00 )
   END_RUNG
   // the same network as SCL:
   #wrkCtrlPriority00 := NOT #wrkCtrlPriority40 AND NOT #wrkCtrlPriority30 AND NOT #wrkCtrlPriority20 AND NOT #wrkCtrlPriority10;
END_REGION

REGION Network 25: Signal conditioning — Consolidate the auto or manual state request
   // ▀▀▀▀▀▀▀▀▀▀▀▀▀▀▀▀▀▀▀▀▀▀▀▀▀▀▀▀▀▀▀▀▀▀▀▀▀▀▀▀▀▀▀▀
   // Determine the valve state required by the automatic/manual mode selection:
   // 
   //    1.  If manual mode is active set wrkCtrlAutManOpCl to match the current manual 
   //      mode requested state (ctrl_Man_OpenClose)
   // 
   //    2.  If automatic mode is active set wrkCtrlAutManOpCl to match the current automatic 
   //      mode requested state (ctrl_Aut_OpenClose)
   // ▄▄▄▄▄▄▄▄▄▄▄▄▄▄▄▄▄▄▄▄▄▄▄▄▄▄▄▄▄▄▄▄▄▄▄▄▄▄▄▄▄▄▄▄
   RUNG wire#powerrail
      Contact( #DYNAMIC_DATA.mode_AutMan )
      Contact( #DYNAMIC_DATA.ctrl_Aut_OpenClose )
      wire#w1
      Coil( #wrkCtrlAutManOpCl )
   END_RUNG
   RUNG wire#powerrail
      I_Contact( #DYNAMIC_DATA.mode_AutMan )
      Contact( #DYNAMIC_DATA.ctrl_Man_OpenClose )
   END_RUNG wire#w1
   // the same network as SCL:
   #wrkCtrlAutManOpCl := (#DYNAMIC_DATA.mode_AutMan AND #DYNAMIC_DATA.ctrl_Aut_OpenClose) OR (NOT #DYNAMIC_DATA.mode_AutMan AND #DYNAMIC_DATA.ctrl_Man_OpenClose);
END_REGION

REGION Network 26: Control — Evaluate priority signals and set open/close request (Priority 40)
   // ▀▀▀▀▀▀▀▀▀▀▀▀▀▀▀▀▀▀▀▀▀▀▀▀▀▀▀▀▀▀▀▀▀▀▀▀▀▀▀▀▀▀▀▀
   // If  a priority 40 (safety) condition is active, set the valve to the deenergised 
   // state:
   // 
   //    •   If the valve is normally open (CONFIG_NO_NC = 1), the deenergised state is open
   // 
   //    •   If the valve is normally closed (CONFIG_NO_NC = 0), the deenergised state is closed
   // ▄▄▄▄▄▄▄▄▄▄▄▄▄▄▄▄▄▄▄▄▄▄▄▄▄▄▄▄▄▄▄▄▄▄▄▄▄▄▄▄▄▄▄▄
   RUNG wire#powerrail
      Contact( #wrkCtrlPriority40 )
      wire#w1
      Contact( #STATIC_DATA.CONFIG_NO_NC )
      S_Coil( #DYNAMIC_DATA."$ctrl_OpenClose" )
   END_RUNG
   RUNG wire#w1
      I_Contact( #STATIC_DATA.CONFIG_NO_NC )
      R_Coil( #DYNAMIC_DATA."$ctrl_OpenClose" )
   END_RUNG
   // the same network as SCL:
   IF #wrkCtrlPriority40 AND #STATIC_DATA.CONFIG_NO_NC THEN #DYNAMIC_DATA."$ctrl_OpenClose" := TRUE; END_IF;
   IF #wrkCtrlPriority40 AND NOT #STATIC_DATA.CONFIG_NO_NC THEN
       #DYNAMIC_DATA."$ctrl_OpenClose" := FALSE;
   END_IF;
END_REGION

REGION Network 27: Control — Evaluate priority signals and set open/close request (Priority 30)
   // ▀▀▀▀▀▀▀▀▀▀▀▀▀▀▀▀▀▀▀▀▀▀▀▀▀▀▀▀▀▀▀▀▀▀▀▀▀▀▀▀▀▀▀▀
   // If  a priority 30 (trip) condition is active, set the valve to the required state:
   // 
   //    •   If the TRIP state is open (CONFIG_TRIP_OP_CL = 1) set the valve to be open
   // 
   //    •   f the TRIP state is closed (CONFIG_TRIP_OP_CL = 0) set the valve to be closed
   // ▄▄▄▄▄▄▄▄▄▄▄▄▄▄▄▄▄▄▄▄▄▄▄▄▄▄▄▄▄▄▄▄▄▄▄▄▄▄▄▄▄▄▄▄
   RUNG wire#powerrail
      Contact( #wrkCtrlPriority30 )
      wire#w1
      Contact( #STATIC_DATA.CONFIG_TRIP_OP_CL )
      S_Coil( #DYNAMIC_DATA."$ctrl_OpenClose" )
   END_RUNG
   RUNG wire#w1
      I_Contact( #STATIC_DATA.CONFIG_TRIP_OP_CL )
      R_Coil( #DYNAMIC_DATA."$ctrl_OpenClose" )
   END_RUNG
   // the same network as SCL:
   IF #wrkCtrlPriority30 AND #STATIC_DATA.CONFIG_TRIP_OP_CL THEN
       #DYNAMIC_DATA."$ctrl_OpenClose" := TRUE;
   END_IF;
   IF #wrkCtrlPriority30 AND NOT #STATIC_DATA.CONFIG_TRIP_OP_CL THEN
       #DYNAMIC_DATA."$ctrl_OpenClose" := FALSE;
   END_IF;
END_REGION

REGION Network 28: Control — Evaluate priority signals and set open/close request (Priority 20)
   // ▀▀▀▀▀▀▀▀▀▀▀▀▀▀▀▀▀▀▀▀▀▀▀▀▀▀▀▀▀▀▀▀▀▀▀▀▀▀▀▀▀▀▀▀
   // If  a priority 20 (interlock) condition is active, set the valve to the required state:
   // 
   //    •   If the INTERLOCK state is open (CONFIG_ILOCK_OP_CL = 1) set the valve to be open
   // 
   //    •   f the INTERLOCK state is closed (CONFIG_ILOCK_OP_CL = 0) set the valve to be closed
   // ▄▄▄▄▄▄▄▄▄▄▄▄▄▄▄▄▄▄▄▄▄▄▄▄▄▄▄▄▄▄▄▄▄▄▄▄▄▄▄▄▄▄▄▄
   RUNG wire#powerrail
      Contact( #wrkCtrlPriority20 )
      wire#w1
      Contact( #STATIC_DATA.CONFIG_ILOCK_OP_CL )
      S_Coil( #DYNAMIC_DATA."$ctrl_OpenClose" )
   END_RUNG
   RUNG wire#w1
      I_Contact( #STATIC_DATA.CONFIG_ILOCK_OP_CL )
      R_Coil( #DYNAMIC_DATA."$ctrl_OpenClose" )
   END_RUNG
   // the same network as SCL:
   IF #wrkCtrlPriority20 AND #STATIC_DATA.CONFIG_ILOCK_OP_CL THEN
       #DYNAMIC_DATA."$ctrl_OpenClose" := TRUE;
   END_IF;
   IF #wrkCtrlPriority20 AND NOT #STATIC_DATA.CONFIG_ILOCK_OP_CL THEN
       #DYNAMIC_DATA."$ctrl_OpenClose" := FALSE;
   END_IF;
END_REGION

REGION Network 29: Control — Evaluate priority signals and set open/close request (Priority 10)
   // ▀▀▀▀▀▀▀▀▀▀▀▀▀▀▀▀▀▀▀▀▀▀▀▀▀▀▀▀▀▀▀▀▀▀▀▀▀▀▀▀▀▀▀▀
   // If  a priority 10 (permissive) condition is active, set the valve to the required state:
   // 
   // 
   // PERMITTED STATE IS OPEN — CONDITIONS:
   // 
   //    •   If the Permitted state is open and Aut/Man request is for open, 
   //      set the valve to be open [Branch 1]
   // 
   //    •   If the Permitted state is open and Aut/Man request is for closed, and the current
   //      valve output matches this state (closed), set the valve to be closed (maintain the
   //      current state) [Branch 6]
   // 
   //    •   If the Permitted state is open and Aut/Man request is for closed, and the current
   //      valve output matches the open state, set the valve to be open (override the
   //      auto/man request [Branch 2]
   // 
   // PERMITTED STATE IS CLOSED — CONDITIONS:
   // 
   //    •   If the Permitted state is closed and Aut/Man request is for closed,
   //      set the valve to be  closed [Branch 4]
   // 
   //    •   If the Permitted state is closed and Aut/Man request is for open, and the current
   //      valve output matches this state (open), set the valve to be open (maintain the
   //      current state) [Branch 3]
   // 
   //    •   If the Permitted state is closed and Aut/Man request is for open, and the current
   //      valve output matches the closed state, set the valve to be closed (override the
   //      auto/man request [Branch 5]
   // ▄▄▄▄▄▄▄▄▄▄▄▄▄▄▄▄▄▄▄▄▄▄▄▄▄▄▄▄▄▄▄▄▄▄▄▄▄▄▄▄▄▄▄▄
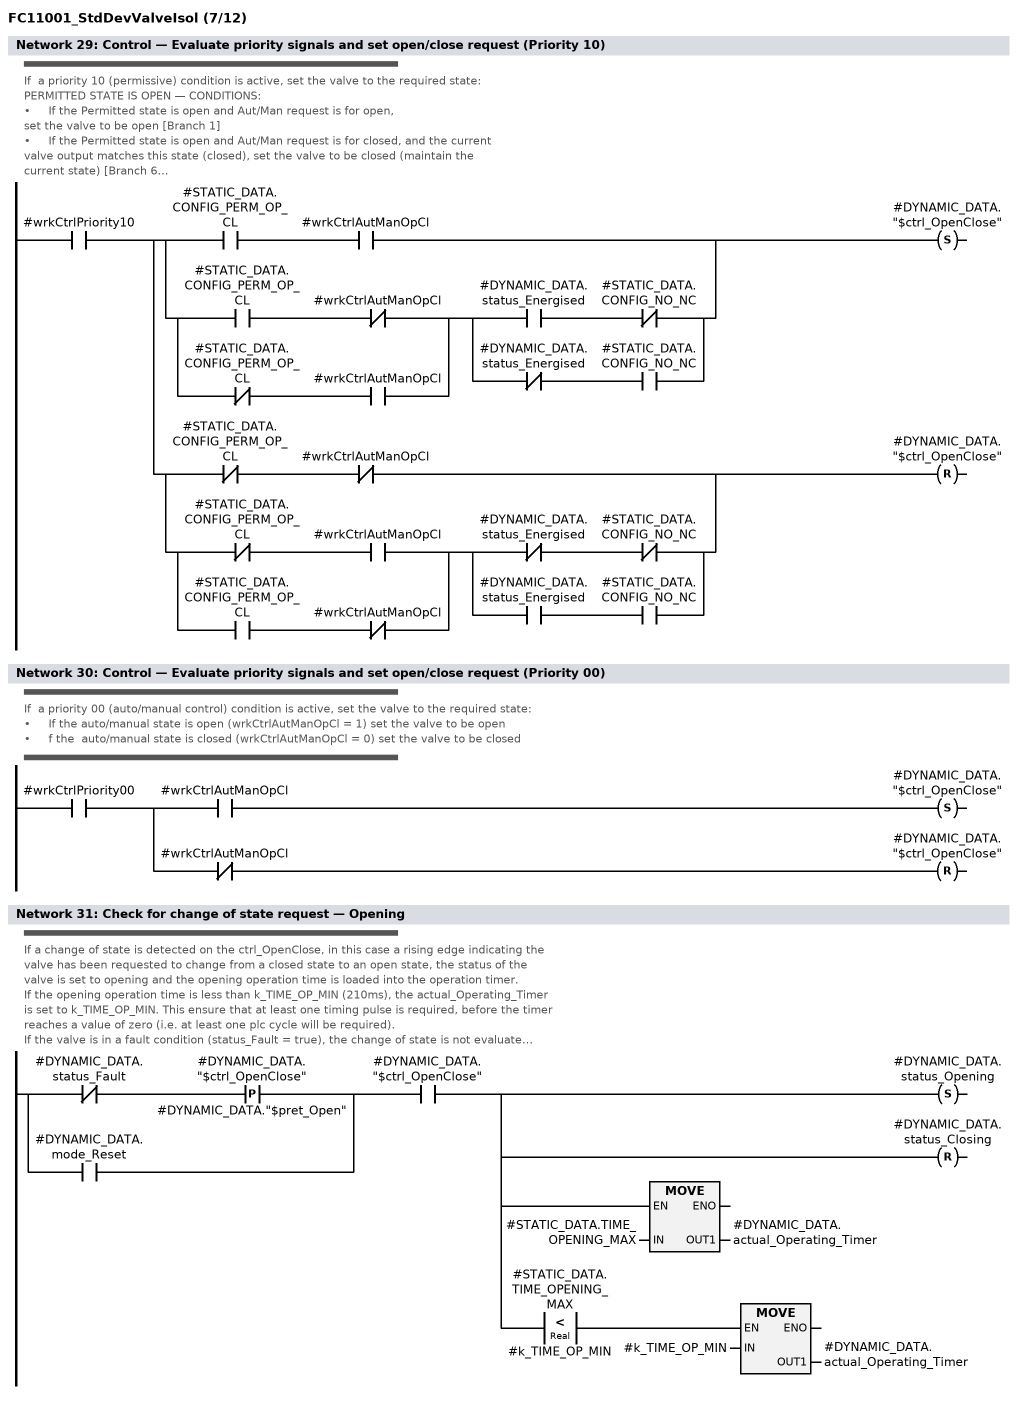
   RUNG wire#powerrail
      Contact( #wrkCtrlPriority10 )
      wire#w1
      Contact( #STATIC_DATA.CONFIG_PERM_OP_CL )
      Contact( #wrkCtrlAutManOpCl )
      wire#w2
      S_Coil( #DYNAMIC_DATA."$ctrl_OpenClose" )
   END_RUNG
   RUNG wire#w1
      Contact( #STATIC_DATA.CONFIG_PERM_OP_CL )
      I_Contact( #wrkCtrlAutManOpCl )
      wire#w3
      Contact( #DYNAMIC_DATA.status_Energised )
      I_Contact( #STATIC_DATA.CONFIG_NO_NC )
   END_RUNG wire#w2
   RUNG wire#w1
      I_Contact( #STATIC_DATA.CONFIG_PERM_OP_CL )
      Contact( #wrkCtrlAutManOpCl )
   END_RUNG wire#w3
   RUNG wire#w3
      I_Contact( #DYNAMIC_DATA.status_Energised )
      Contact( #STATIC_DATA.CONFIG_NO_NC )
   END_RUNG wire#w2
   RUNG wire#w1
      I_Contact( #STATIC_DATA.CONFIG_PERM_OP_CL )
      I_Contact( #wrkCtrlAutManOpCl )
      wire#w4
      R_Coil( #DYNAMIC_DATA."$ctrl_OpenClose" )
   END_RUNG
   RUNG wire#w1
      I_Contact( #STATIC_DATA.CONFIG_PERM_OP_CL )
      Contact( #wrkCtrlAutManOpCl )
      wire#w5
      I_Contact( #DYNAMIC_DATA.status_Energised )
      I_Contact( #STATIC_DATA.CONFIG_NO_NC )
   END_RUNG wire#w4
   RUNG wire#w1
      Contact( #STATIC_DATA.CONFIG_PERM_OP_CL )
      I_Contact( #wrkCtrlAutManOpCl )
   END_RUNG wire#w5
   RUNG wire#w5
      Contact( #DYNAMIC_DATA.status_Energised )
      Contact( #STATIC_DATA.CONFIG_NO_NC )
   END_RUNG wire#w4
   // the same network as SCL:
   IF #wrkCtrlPriority10 AND ((#STATIC_DATA.CONFIG_PERM_OP_CL AND #wrkCtrlAutManOpCl) OR (((#STATIC_DATA.CONFIG_PERM_OP_CL AND NOT #wrkCtrlAutManOpCl) OR (NOT #STATIC_DATA.CONFIG_PERM_OP_CL AND #wrkCtrlAutManOpCl)) AND ((#DYNAMIC_DATA.status_Energised AND NOT #STATIC_DATA.CONFIG_NO_NC) OR (NOT #DYNAMIC_DATA.status_Energised AND #STATIC_DATA.CONFIG_NO_NC)))) THEN
       #DYNAMIC_DATA."$ctrl_OpenClose" := TRUE;
   END_IF;
   IF #wrkCtrlPriority10 AND ((NOT #STATIC_DATA.CONFIG_PERM_OP_CL AND NOT #wrkCtrlAutManOpCl) OR (((NOT #STATIC_DATA.CONFIG_PERM_OP_CL AND #wrkCtrlAutManOpCl) OR (#STATIC_DATA.CONFIG_PERM_OP_CL AND NOT #wrkCtrlAutManOpCl)) AND ((NOT #DYNAMIC_DATA.status_Energised AND NOT #STATIC_DATA.CONFIG_NO_NC) OR (#DYNAMIC_DATA.status_Energised AND #STATIC_DATA.CONFIG_NO_NC)))) THEN
       #DYNAMIC_DATA."$ctrl_OpenClose" := FALSE;
   END_IF;
END_REGION

REGION Network 30: Control — Evaluate priority signals and set open/close request (Priority 00)
   // ▀▀▀▀▀▀▀▀▀▀▀▀▀▀▀▀▀▀▀▀▀▀▀▀▀▀▀▀▀▀▀▀▀▀▀▀▀▀▀▀▀▀▀▀
   // If  a priority 00 (auto/manual control) condition is active, set the valve to the required state:
   // 
   //    •   If the auto/manual state is open (wrkCtrlAutManOpCl = 1) set the valve to be open
   // 
   //    •   f the  auto/manual state is closed (wrkCtrlAutManOpCl = 0) set the valve to be closed
   // ▄▄▄▄▄▄▄▄▄▄▄▄▄▄▄▄▄▄▄▄▄▄▄▄▄▄▄▄▄▄▄▄▄▄▄▄▄▄▄▄▄▄▄▄
   RUNG wire#powerrail
      Contact( #wrkCtrlPriority00 )
      wire#w1
      Contact( #wrkCtrlAutManOpCl )
      S_Coil( #DYNAMIC_DATA."$ctrl_OpenClose" )
   END_RUNG
   RUNG wire#w1
      I_Contact( #wrkCtrlAutManOpCl )
      R_Coil( #DYNAMIC_DATA."$ctrl_OpenClose" )
   END_RUNG
   // the same network as SCL:
   IF #wrkCtrlPriority00 AND #wrkCtrlAutManOpCl THEN #DYNAMIC_DATA."$ctrl_OpenClose" := TRUE; END_IF;
   IF #wrkCtrlPriority00 AND NOT #wrkCtrlAutManOpCl THEN #DYNAMIC_DATA."$ctrl_OpenClose" := FALSE; END_IF;
END_REGION

REGION Network 31: Check for change of state request — Opening
   // ▀▀▀▀▀▀▀▀▀▀▀▀▀▀▀▀▀▀▀▀▀▀▀▀▀▀▀▀▀▀▀▀▀▀▀▀▀▀▀▀▀▀▀▀
   // If a change of state is detected on the ctrl_OpenClose, in this case a rising edge indicating the
   // valve has been requested to change from a closed state to an open state, the status of the
   // valve is set to opening and the opening operation time is loaded into the operation timer.
   // 
   // If the opening operation time is less than k_TIME_OP_MIN (210ms), the actual_Operating_Timer 
   // is set to k_TIME_OP_MIN. This ensure that at least one timing pulse is required, before the timer 
   // reaches a value of zero (i.e. at least one plc cycle will be required).
   // 
   // If the valve is in a fault condition (status_Fault = true), the change of state is not evaluated
   // until the fault condition has cleared
   // 
   // Note: the timer is also triggered if the Reset signal is received and the valve is requested open.
   // ▄▄▄▄▄▄▄▄▄▄▄▄▄▄▄▄▄▄▄▄▄▄▄▄▄▄▄▄▄▄▄▄▄▄▄▄▄▄▄▄▄▄▄▄
   RUNG wire#powerrail
      I_Contact( #DYNAMIC_DATA.status_Fault )
      P_Contact(operand := #DYNAMIC_DATA."$ctrl_OpenClose", bit := #DYNAMIC_DATA."$pret_Open")
      wire#w1
      Contact( #DYNAMIC_DATA."$ctrl_OpenClose" )
      wire#w2
      S_Coil( #DYNAMIC_DATA.status_Opening )
   END_RUNG
   RUNG wire#powerrail
      Contact( #DYNAMIC_DATA.mode_Reset )
   END_RUNG wire#w1
   RUNG wire#w2
      R_Coil( #DYNAMIC_DATA.status_Closing )
   END_RUNG
   RUNG wire#w2
      Move(in := #STATIC_DATA.TIME_OPENING_MAX, out1 => #DYNAMIC_DATA.actual_Operating_Timer)
   END_RUNG
   RUNG wire#w2
      { S7_Templates := "SrcType := Real" } LT_Contact(in1 := #STATIC_DATA.TIME_OPENING_MAX, in2 := #k_TIME_OP_MIN)
      Move(in := #k_TIME_OP_MIN, out1 => #DYNAMIC_DATA.actual_Operating_Timer)
   END_RUNG
   // the same network as SCL:
   #_w1 := NOT #DYNAMIC_DATA.status_Fault AND #DYNAMIC_DATA."$ctrl_OpenClose" AND NOT #DYNAMIC_DATA."$pret_Open";   // rising edge of #DYNAMIC_DATA."$ctrl_OpenClose"
   #DYNAMIC_DATA."$pret_Open" := #DYNAMIC_DATA."$ctrl_OpenClose";
   #_w2 := (#_w1 OR #DYNAMIC_DATA.mode_Reset) AND #DYNAMIC_DATA."$ctrl_OpenClose";
   IF #_w2 THEN
       #DYNAMIC_DATA.status_Opening := TRUE;
       #DYNAMIC_DATA.status_Closing := FALSE;
       #DYNAMIC_DATA.actual_Operating_Timer := #STATIC_DATA.TIME_OPENING_MAX;
   END_IF;
   IF #_w2 AND (#STATIC_DATA.TIME_OPENING_MAX < #k_TIME_OP_MIN) THEN
       #DYNAMIC_DATA.actual_Operating_Timer := #k_TIME_OP_MIN;
   END_IF;
END_REGION

REGION Network 32: Check for change of state request — Closing
   // ▀▀▀▀▀▀▀▀▀▀▀▀▀▀▀▀▀▀▀▀▀▀▀▀▀▀▀▀▀▀▀▀▀▀▀▀▀▀▀▀▀▀▀▀
   // If a change of state is detected on the ctrl_OpenClose, in this case a falling edge indicating the
   // valve has been requested to change from an open state to a closed state, the status of the
   // valve is set to closing and the closing operation time is loaded into the operation timer.
   // 
   // If the closing operation time is less than k_TIME_OP_MIN (210ms), the actual_Operating_Timer 
   // is set to k_TIME_OP_MIN. This ensure that at least one timing pulse is required, before the timer 
   // reaches a value of zero (i.e. at least one plc cycle will be required).
   // 
   // If the valve is in a fault condition (status_Fault = true), the change of state is not evaluated
   // until the fault condition has cleared
   // 
   // Note: the timer is also triggered if the Reset signal is received and the valve is requested closed.
   // ▄▄▄▄▄▄▄▄▄▄▄▄▄▄▄▄▄▄▄▄▄▄▄▄▄▄▄▄▄▄▄▄▄▄▄▄▄▄▄▄▄▄▄▄
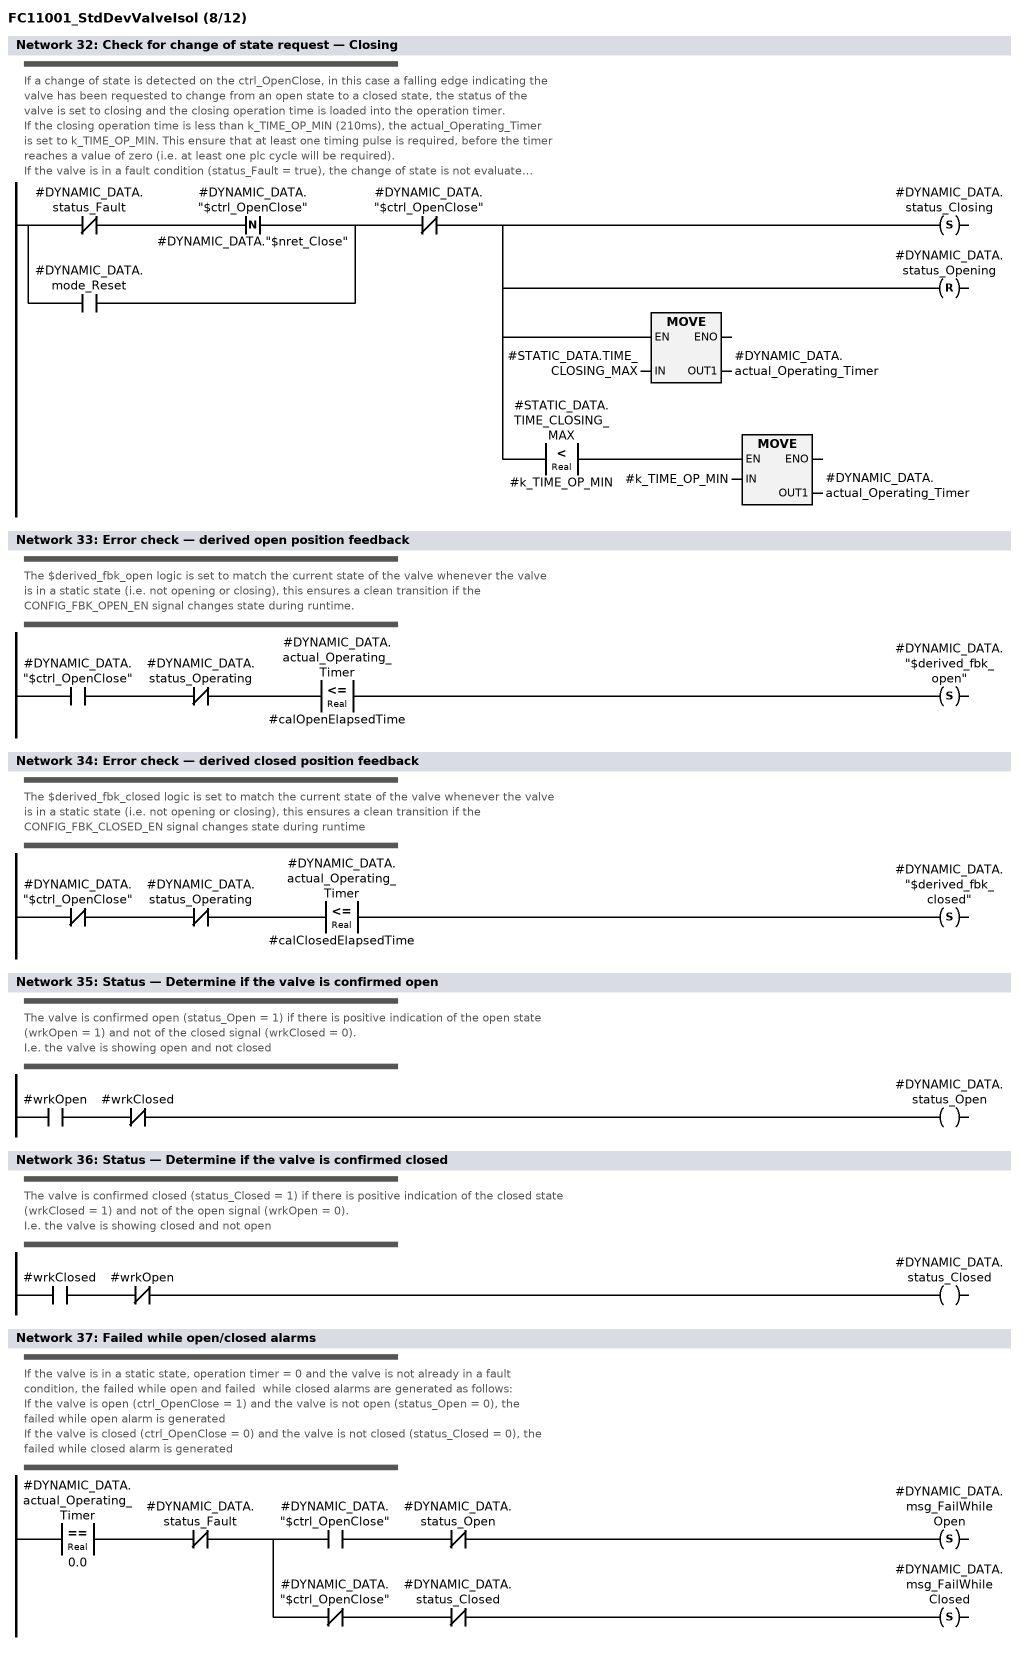
   RUNG wire#powerrail
      I_Contact( #DYNAMIC_DATA.status_Fault )
      N_Contact(operand := #DYNAMIC_DATA."$ctrl_OpenClose", bit := #DYNAMIC_DATA."$nret_Close")
      wire#w1
      I_Contact( #DYNAMIC_DATA."$ctrl_OpenClose" )
      wire#w2
      S_Coil( #DYNAMIC_DATA.status_Closing )
   END_RUNG
   RUNG wire#powerrail
      Contact( #DYNAMIC_DATA.mode_Reset )
   END_RUNG wire#w1
   RUNG wire#w2
      R_Coil( #DYNAMIC_DATA.status_Opening )
   END_RUNG
   RUNG wire#w2
      Move(in := #STATIC_DATA.TIME_CLOSING_MAX, out1 => #DYNAMIC_DATA.actual_Operating_Timer)
   END_RUNG
   RUNG wire#w2
      { S7_Templates := "SrcType := Real" } LT_Contact(in1 := #STATIC_DATA.TIME_CLOSING_MAX, in2 := #k_TIME_OP_MIN)
      Move(in := #k_TIME_OP_MIN, out1 => #DYNAMIC_DATA.actual_Operating_Timer)
   END_RUNG
   // the same network as SCL:
   #_w1 := NOT #DYNAMIC_DATA.status_Fault AND NOT #DYNAMIC_DATA."$ctrl_OpenClose" AND #DYNAMIC_DATA."$nret_Close";   // falling edge of #DYNAMIC_DATA."$ctrl_OpenClose"
   #DYNAMIC_DATA."$nret_Close" := #DYNAMIC_DATA."$ctrl_OpenClose";
   #_w2 := (#_w1 OR #DYNAMIC_DATA.mode_Reset) AND NOT #DYNAMIC_DATA."$ctrl_OpenClose";
   IF #_w2 THEN
       #DYNAMIC_DATA.status_Closing := TRUE;
       #DYNAMIC_DATA.status_Opening := FALSE;
       #DYNAMIC_DATA.actual_Operating_Timer := #STATIC_DATA.TIME_CLOSING_MAX;
   END_IF;
   IF #_w2 AND (#STATIC_DATA.TIME_CLOSING_MAX < #k_TIME_OP_MIN) THEN
       #DYNAMIC_DATA.actual_Operating_Timer := #k_TIME_OP_MIN;
   END_IF;
END_REGION

REGION Network 33: Error check — derived open position feedback
   // ▀▀▀▀▀▀▀▀▀▀▀▀▀▀▀▀▀▀▀▀▀▀▀▀▀▀▀▀▀▀▀▀▀▀▀▀▀▀▀▀▀▀▀▀
   // The $derived_fbk_open logic is set to match the current state of the valve whenever the valve
   // is in a static state (i.e. not opening or closing), this ensures a clean transition if the 
   // CONFIG_FBK_OPEN_EN signal changes state during runtime.
   // ▄▄▄▄▄▄▄▄▄▄▄▄▄▄▄▄▄▄▄▄▄▄▄▄▄▄▄▄▄▄▄▄▄▄▄▄▄▄▄▄▄▄▄▄
   RUNG wire#powerrail
      Contact( #DYNAMIC_DATA."$ctrl_OpenClose" )
      I_Contact( #DYNAMIC_DATA.status_Operating )
      { S7_Templates := "SrcType := Real" } LE_Contact(in1 := #DYNAMIC_DATA.actual_Operating_Timer, in2 := #calOpenElapsedTime)
      S_Coil( #DYNAMIC_DATA."$derived_fbk_open" )
   END_RUNG
   // the same network as SCL:
   IF #DYNAMIC_DATA."$ctrl_OpenClose" AND NOT #DYNAMIC_DATA.status_Operating AND (#DYNAMIC_DATA.actual_Operating_Timer <= #calOpenElapsedTime) THEN
       #DYNAMIC_DATA."$derived_fbk_open" := TRUE;
   END_IF;
END_REGION

REGION Network 34: Error check — derived closed position feedback
   // ▀▀▀▀▀▀▀▀▀▀▀▀▀▀▀▀▀▀▀▀▀▀▀▀▀▀▀▀▀▀▀▀▀▀▀▀▀▀▀▀▀▀▀▀
   // The $derived_fbk_closed logic is set to match the current state of the valve whenever the valve
   // is in a static state (i.e. not opening or closing), this ensures a clean transition if the 
   // CONFIG_FBK_CLOSED_EN signal changes state during runtime
   // ▄▄▄▄▄▄▄▄▄▄▄▄▄▄▄▄▄▄▄▄▄▄▄▄▄▄▄▄▄▄▄▄▄▄▄▄▄▄▄▄▄▄▄▄
   RUNG wire#powerrail
      I_Contact( #DYNAMIC_DATA."$ctrl_OpenClose" )
      I_Contact( #DYNAMIC_DATA.status_Operating )
      { S7_Templates := "SrcType := Real" } LE_Contact(in1 := #DYNAMIC_DATA.actual_Operating_Timer, in2 := #calClosedElapsedTime)
      S_Coil( #DYNAMIC_DATA."$derived_fbk_closed" )
   END_RUNG
   // the same network as SCL:
   IF NOT #DYNAMIC_DATA."$ctrl_OpenClose" AND NOT #DYNAMIC_DATA.status_Operating AND (#DYNAMIC_DATA.actual_Operating_Timer <= #calClosedElapsedTime) THEN
       #DYNAMIC_DATA."$derived_fbk_closed" := TRUE;
   END_IF;
END_REGION

REGION Network 35: Status — Determine if the valve is confirmed open
   // ▀▀▀▀▀▀▀▀▀▀▀▀▀▀▀▀▀▀▀▀▀▀▀▀▀▀▀▀▀▀▀▀▀▀▀▀▀▀▀▀▀▀▀▀
   // The valve is confirmed open (status_Open = 1) if there is positive indication of the open state 
   // (wrkOpen = 1) and not of the closed signal (wrkClosed = 0). 
   // 
   // I.e. the valve is showing open and not closed
   // ▄▄▄▄▄▄▄▄▄▄▄▄▄▄▄▄▄▄▄▄▄▄▄▄▄▄▄▄▄▄▄▄▄▄▄▄▄▄▄▄▄▄▄▄
   RUNG wire#powerrail
      Contact( #wrkOpen )
      I_Contact( #wrkClosed )
      Coil( #DYNAMIC_DATA.status_Open )
   END_RUNG
   // the same network as SCL:
   #DYNAMIC_DATA.status_Open := #wrkOpen AND NOT #wrkClosed;
END_REGION

REGION Network 36: Status — Determine if the valve is confirmed closed
   // ▀▀▀▀▀▀▀▀▀▀▀▀▀▀▀▀▀▀▀▀▀▀▀▀▀▀▀▀▀▀▀▀▀▀▀▀▀▀▀▀▀▀▀▀
   // The valve is confirmed closed (status_Closed = 1) if there is positive indication of the closed state 
   // (wrkClosed = 1) and not of the open signal (wrkOpen = 0). 
   // 
   // I.e. the valve is showing closed and not open
   // ▄▄▄▄▄▄▄▄▄▄▄▄▄▄▄▄▄▄▄▄▄▄▄▄▄▄▄▄▄▄▄▄▄▄▄▄▄▄▄▄▄▄▄▄
   RUNG wire#powerrail
      Contact( #wrkClosed )
      I_Contact( #wrkOpen )
      Coil( #DYNAMIC_DATA.status_Closed )
   END_RUNG
   // the same network as SCL:
   #DYNAMIC_DATA.status_Closed := #wrkClosed AND NOT #wrkOpen;
END_REGION

REGION Network 37: Failed while open/closed alarms
   // ▀▀▀▀▀▀▀▀▀▀▀▀▀▀▀▀▀▀▀▀▀▀▀▀▀▀▀▀▀▀▀▀▀▀▀▀▀▀▀▀▀▀▀▀
   // If the valve is in a static state, operation timer = 0 and the valve is not already in a fault
   // condition, the failed while open and failed  while closed alarms are generated as follows:
   // 
   // If the valve is open (ctrl_OpenClose = 1) and the valve is not open (status_Open = 0), the 
   // failed while open alarm is generated
   // 
   // If the valve is closed (ctrl_OpenClose = 0) and the valve is not closed (status_Closed = 0), the 
   // failed while closed alarm is generated
   // ▄▄▄▄▄▄▄▄▄▄▄▄▄▄▄▄▄▄▄▄▄▄▄▄▄▄▄▄▄▄▄▄▄▄▄▄▄▄▄▄▄▄▄▄
   RUNG wire#powerrail
      { S7_Templates := "SrcType := Real" } EQ_Contact(in1 := #DYNAMIC_DATA.actual_Operating_Timer, in2 := 0.0)
      I_Contact( #DYNAMIC_DATA.status_Fault )
      wire#w1
      Contact( #DYNAMIC_DATA."$ctrl_OpenClose" )
      I_Contact( #DYNAMIC_DATA.status_Open )
      S_Coil( #DYNAMIC_DATA.msg_FailWhileOpen )
   END_RUNG
   RUNG wire#w1
      I_Contact( #DYNAMIC_DATA."$ctrl_OpenClose" )
      I_Contact( #DYNAMIC_DATA.status_Closed )
      S_Coil( #DYNAMIC_DATA.msg_FailWhileClosed )
   END_RUNG
   // the same network as SCL:
   #_w1 := (#DYNAMIC_DATA.actual_Operating_Timer = 0.0) AND NOT #DYNAMIC_DATA.status_Fault;
   IF #_w1 AND #DYNAMIC_DATA."$ctrl_OpenClose" AND NOT #DYNAMIC_DATA.status_Open THEN
       #DYNAMIC_DATA.msg_FailWhileOpen := TRUE;
   END_IF;
   IF #_w1 AND NOT #DYNAMIC_DATA."$ctrl_OpenClose" AND NOT #DYNAMIC_DATA.status_Closed THEN
       #DYNAMIC_DATA.msg_FailWhileClosed := TRUE;
   END_IF;
END_REGION

REGION Network 38: Operation timer and Failed to open/close alarms
   // ▀▀▀▀▀▀▀▀▀▀▀▀▀▀▀▀▀▀▀▀▀▀▀▀▀▀▀▀▀▀▀▀▀▀▀▀▀▀▀▀▀▀▀▀
   // If the valve is opening or closing, decrement the current operation timer value on each 200ms
   // pulse.
   // 
   // If the timer reaches zero, and the valve is opening, generate the failed to open alarm.
   // 
   // If the timer reaches zero, and the valve is closing, generate the failed to close alarm
   // ▄▄▄▄▄▄▄▄▄▄▄▄▄▄▄▄▄▄▄▄▄▄▄▄▄▄▄▄▄▄▄▄▄▄▄▄▄▄▄▄▄▄▄▄
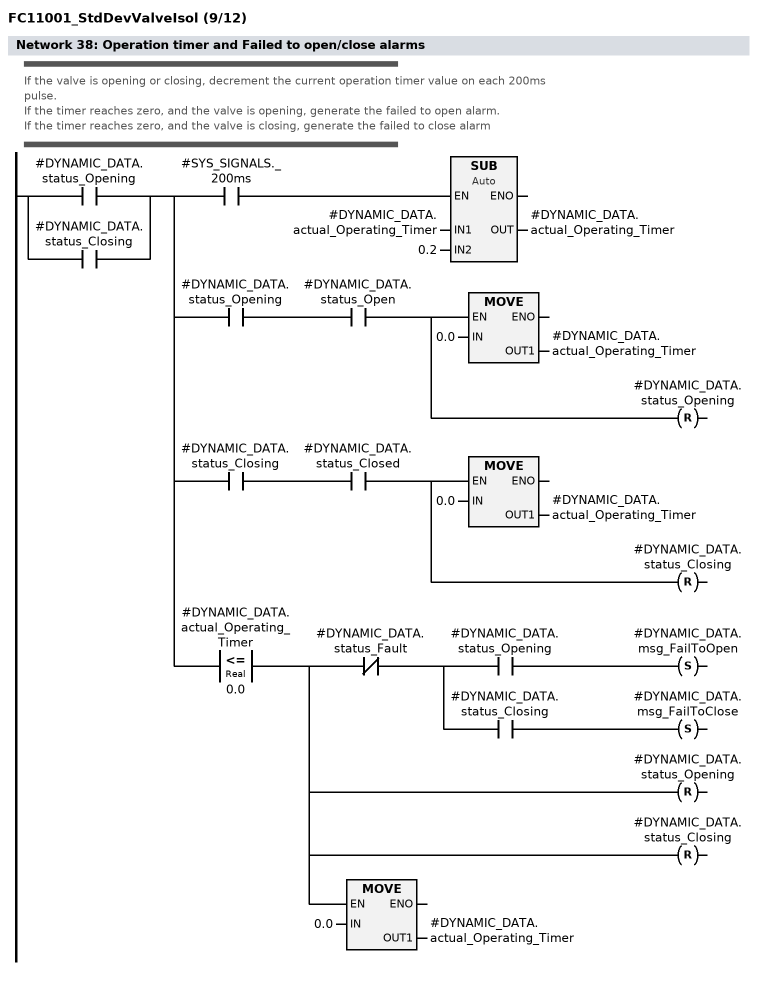
   RUNG wire#powerrail
      Contact( #DYNAMIC_DATA.status_Opening )
      wire#w1
      Contact( #SYS_SIGNALS._200ms )
      Sub(in1 := #DYNAMIC_DATA.actual_Operating_Timer, in2 := 0.2, out => #DYNAMIC_DATA.actual_Operating_Timer)
   END_RUNG
   RUNG wire#powerrail
      Contact( #DYNAMIC_DATA.status_Closing )
   END_RUNG wire#w1
   RUNG wire#w1
      Contact( #DYNAMIC_DATA.status_Opening )
      Contact( #DYNAMIC_DATA.status_Open )
      wire#w2
      Move(in := 0.0, out1 => #DYNAMIC_DATA.actual_Operating_Timer)
   END_RUNG
   RUNG wire#w2
      R_Coil( #DYNAMIC_DATA.status_Opening )
   END_RUNG
   RUNG wire#w1
      Contact( #DYNAMIC_DATA.status_Closing )
      Contact( #DYNAMIC_DATA.status_Closed )
      wire#w3
      Move(in := 0.0, out1 => #DYNAMIC_DATA.actual_Operating_Timer)
   END_RUNG
   RUNG wire#w3
      R_Coil( #DYNAMIC_DATA.status_Closing )
   END_RUNG
   RUNG wire#w1
      { S7_Templates := "SrcType := Real" } LE_Contact(in1 := #DYNAMIC_DATA.actual_Operating_Timer, in2 := 0.0)
      wire#w4
      I_Contact( #DYNAMIC_DATA.status_Fault )
      wire#w5
      Contact( #DYNAMIC_DATA.status_Opening )
      S_Coil( #DYNAMIC_DATA.msg_FailToOpen )
   END_RUNG
   RUNG wire#w5
      Contact( #DYNAMIC_DATA.status_Closing )
      S_Coil( #DYNAMIC_DATA.msg_FailToClose )
   END_RUNG
   RUNG wire#w4
      R_Coil( #DYNAMIC_DATA.status_Opening )
   END_RUNG
   RUNG wire#w4
      R_Coil( #DYNAMIC_DATA.status_Closing )
   END_RUNG
   RUNG wire#w4
      Move(in := 0.0, out1 => #DYNAMIC_DATA.actual_Operating_Timer)
   END_RUNG
   // the same network as SCL:
   #_w1 := #DYNAMIC_DATA.status_Opening OR #DYNAMIC_DATA.status_Closing;
   IF #_w1 AND #SYS_SIGNALS._200ms THEN
       #DYNAMIC_DATA.actual_Operating_Timer := #DYNAMIC_DATA.actual_Operating_Timer - 0.2;
   END_IF;
   IF #_w1 AND #DYNAMIC_DATA.status_Opening AND #DYNAMIC_DATA.status_Open THEN
       #DYNAMIC_DATA.actual_Operating_Timer := 0.0;
       #DYNAMIC_DATA.status_Opening := FALSE;
   END_IF;
   IF #_w1 AND #DYNAMIC_DATA.status_Closing AND #DYNAMIC_DATA.status_Closed THEN
       #DYNAMIC_DATA.actual_Operating_Timer := 0.0;
       #DYNAMIC_DATA.status_Closing := FALSE;
   END_IF;
   #_w2 := #_w1 AND (#DYNAMIC_DATA.actual_Operating_Timer <= 0.0);
   #_w3 := #_w2 AND NOT #DYNAMIC_DATA.status_Fault;
   IF #_w3 AND #DYNAMIC_DATA.status_Opening THEN #DYNAMIC_DATA.msg_FailToOpen := TRUE; END_IF;
   IF #_w3 AND #DYNAMIC_DATA.status_Closing THEN #DYNAMIC_DATA.msg_FailToClose := TRUE; END_IF;
   IF #_w2 THEN
       #DYNAMIC_DATA.status_Opening := FALSE;
       #DYNAMIC_DATA.status_Closing := FALSE;
       #DYNAMIC_DATA.actual_Operating_Timer := 0.0;
   END_IF;
END_REGION

REGION Network 39: Calculate last operation timer value
   // ▀▀▀▀▀▀▀▀▀▀▀▀▀▀▀▀▀▀▀▀▀▀▀▀▀▀▀▀▀▀▀▀▀▀▀▀▀▀▀▀▀▀▀▀
   // Stores that last good operation timer elapsed time, this is the elapsed value of the 
   // actual_Operating_Timer when the valve achieved the correct position. The result is subtracted
   // from the TIME_OPENING/CLOSING_MAX value to give the true time to achieve position. The result
   // is stored in actual_Last_Op_Time
   // 
   // If the valve were opening, then actual_Last_Op_Time is calculated as follows:
   // 
   // ┌─────────────────────────────────┐
   // │actual_Last_Op_Time = TIME_OPENING_MAX ─ actual_Operating_Timer   │
   // └─────────────────────────────────┘
   // 
   // If the valve were closing, then actual_Last_Op_Time is calculated as follows:
   // 
   // ┌─────────────────────────────────┐
   // │actual_Last_Op_Time = TIME_CLOSING_MAX ─ actual_Operating_Timer   │
   // └─────────────────────────────────┘
   // 
   // If the valve either fails to open or fails to close,  then actual_Last_Op_Time is set to -1.0 to 
   // indicate a fault state.
   // ▄▄▄▄▄▄▄▄▄▄▄▄▄▄▄▄▄▄▄▄▄▄▄▄▄▄▄▄▄▄▄▄▄▄▄▄▄▄▄▄▄▄▄▄
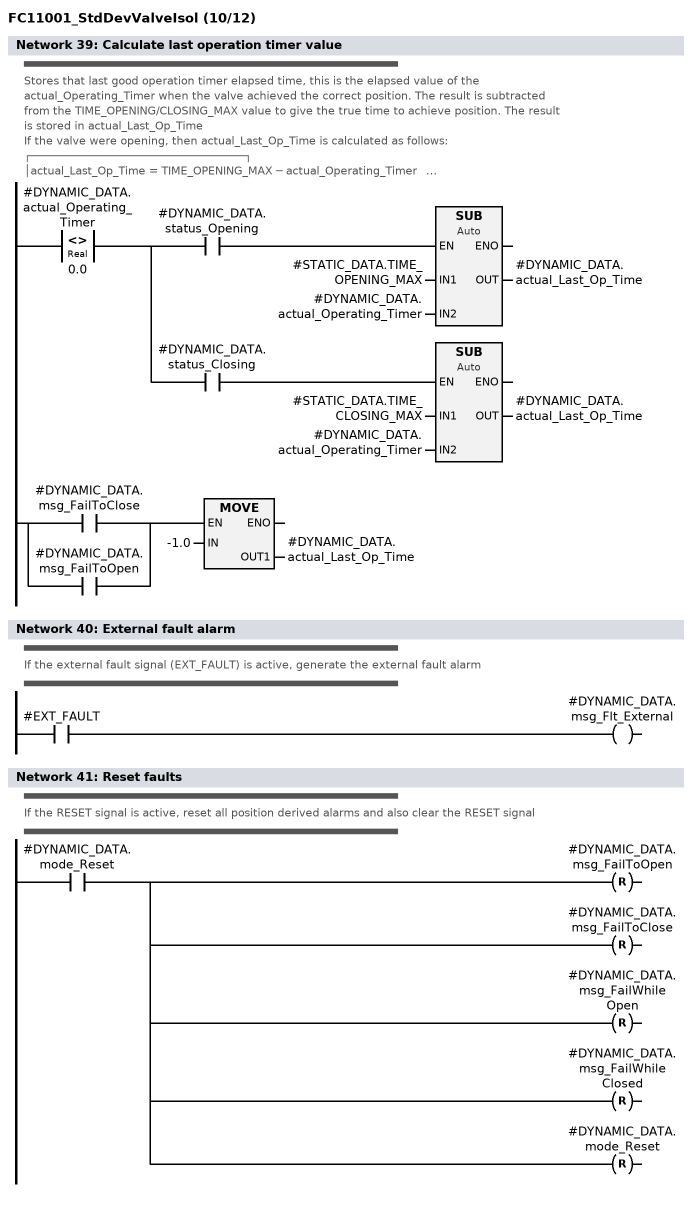
   RUNG wire#powerrail
      { S7_Templates := "SrcType := Real" } NE_Contact(in1 := #DYNAMIC_DATA.actual_Operating_Timer, in2 := 0.0)
      wire#w1
      Contact( #DYNAMIC_DATA.status_Opening )
      Sub(in1 := #STATIC_DATA.TIME_OPENING_MAX, in2 := #DYNAMIC_DATA.actual_Operating_Timer, out => #DYNAMIC_DATA.actual_Last_Op_Time)
   END_RUNG
   RUNG wire#w1
      Contact( #DYNAMIC_DATA.status_Closing )
      Sub(in1 := #STATIC_DATA.TIME_CLOSING_MAX, in2 := #DYNAMIC_DATA.actual_Operating_Timer, out => #DYNAMIC_DATA.actual_Last_Op_Time)
   END_RUNG
   RUNG wire#powerrail
      Contact( #DYNAMIC_DATA.msg_FailToClose )
      wire#w2
      Move(in := -1.0, out1 => #DYNAMIC_DATA.actual_Last_Op_Time)
   END_RUNG
   RUNG wire#powerrail
      Contact( #DYNAMIC_DATA.msg_FailToOpen )
   END_RUNG wire#w2
   // the same network as SCL:
   #_w1 := #DYNAMIC_DATA.actual_Operating_Timer <> 0.0;
   IF #_w1 AND #DYNAMIC_DATA.status_Opening THEN
       #DYNAMIC_DATA.actual_Last_Op_Time := #STATIC_DATA.TIME_OPENING_MAX - #DYNAMIC_DATA.actual_Operating_Timer;
   END_IF;
   IF #_w1 AND #DYNAMIC_DATA.status_Closing THEN
       #DYNAMIC_DATA.actual_Last_Op_Time := #STATIC_DATA.TIME_CLOSING_MAX - #DYNAMIC_DATA.actual_Operating_Timer;
   END_IF;
   IF #DYNAMIC_DATA.msg_FailToClose OR #DYNAMIC_DATA.msg_FailToOpen THEN
       #DYNAMIC_DATA.actual_Last_Op_Time := -1.0;
   END_IF;
END_REGION

REGION Network 40: External fault alarm
   // ▀▀▀▀▀▀▀▀▀▀▀▀▀▀▀▀▀▀▀▀▀▀▀▀▀▀▀▀▀▀▀▀▀▀▀▀▀▀▀▀▀▀▀▀
   // If the external fault signal (EXT_FAULT) is active, generate the external fault alarm
   // ▄▄▄▄▄▄▄▄▄▄▄▄▄▄▄▄▄▄▄▄▄▄▄▄▄▄▄▄▄▄▄▄▄▄▄▄▄▄▄▄▄▄▄▄
   RUNG wire#powerrail
      Contact( #EXT_FAULT )
      Coil( #DYNAMIC_DATA.msg_Flt_External )
   END_RUNG
   // the same network as SCL:
   #DYNAMIC_DATA.msg_Flt_External := #EXT_FAULT;
END_REGION

REGION Network 41: Reset faults
   // ▀▀▀▀▀▀▀▀▀▀▀▀▀▀▀▀▀▀▀▀▀▀▀▀▀▀▀▀▀▀▀▀▀▀▀▀▀▀▀▀▀▀▀▀
   // If the RESET signal is active, reset all position derived alarms and also clear the RESET signal
   // ▄▄▄▄▄▄▄▄▄▄▄▄▄▄▄▄▄▄▄▄▄▄▄▄▄▄▄▄▄▄▄▄▄▄▄▄▄▄▄▄▄▄▄▄
   RUNG wire#powerrail
      Contact( #DYNAMIC_DATA.mode_Reset )
      wire#w1
      R_Coil( #DYNAMIC_DATA.msg_FailToOpen )
   END_RUNG
   RUNG wire#w1
      R_Coil( #DYNAMIC_DATA.msg_FailToClose )
   END_RUNG
   RUNG wire#w1
      R_Coil( #DYNAMIC_DATA.msg_FailWhileOpen )
   END_RUNG
   RUNG wire#w1
      R_Coil( #DYNAMIC_DATA.msg_FailWhileClosed )
   END_RUNG
   RUNG wire#w1
      R_Coil( #DYNAMIC_DATA.mode_Reset )
   END_RUNG
   // the same network as SCL:
   IF #DYNAMIC_DATA.mode_Reset THEN
       #DYNAMIC_DATA.msg_FailToOpen := FALSE;
       #DYNAMIC_DATA.msg_FailToClose := FALSE;
       #DYNAMIC_DATA.msg_FailWhileOpen := FALSE;
       #DYNAMIC_DATA.msg_FailWhileClosed := FALSE;
       #DYNAMIC_DATA.mode_Reset := FALSE;
   END_IF;
END_REGION

REGION Network 42: Status signals
   // ▀▀▀▀▀▀▀▀▀▀▀▀▀▀▀▀▀▀▀▀▀▀▀▀▀▀▀▀▀▀▀▀▀▀▀▀▀▀▀▀▀▀▀▀
   // The status signals for faults, alarms and warnings are either duplicates of the message signals 
   // (signals beginning with msg_) or logical combinations of them.
   // 
   // The following is a full list of the status signals:
   // 
   //  UT31001_Dy_DevValveIsol (full contents)
   //  ――――――――――――――――――――――――――――――――――――――――――
   //  SIGNAL NAME          FUNCTION                     TYPE
   //  ――――――――――――――――――――――――――――――――――――――――――
   //  status_Operating        STATUS — Valve is changing state           Bool
   //                      (1 = changing state, 0 = fixed state)
   //  status_Fault            STATUS — Valve is in fault              Bool
   //                      (1 = fault present, 0 = healthy)
   //  status_Energised        STATUS — Valve output is on              Bool
   //                      (1 = energised, 0 = deenergised)
   //  status_Aut           STATUS — Automatic mode active           Bool
   //                      (1 = auto mode on, 0 = auto mode off)
   //  status_Man          STATUS — Manual mode active             Bool
   //                      (1 = man mode on, 0 = man mode off)
   //  status_EStop          STATUS — E_STOP safety signal is active         Bool
   //                      (1 = active, 0 = healthy)
   //  status_Trip        STATUS — TRIP signal is active             Bool
   //                      (1 = active, 0 = healthy)
   //  status_Ilock         STATUS — INTERLOCK signal is active            Bool
   //                      (1 = active, 0 = healthy)
   //  status_Perm        STATUS — PERMISSIVE signal is active           Bool
   //                      (1 = active, 0 = healthy)
   //  status_BypassOn        STATUS — Valve is in bypass mode          Bool
   //                      (1 = Simulation mode, 0 = normal)
   //  status_SimOn           STATUS — Valve is in simulation mode               Bool
   //                      (1 = Simulation mode, 0 = normal)
   //  status_RemoteOn       STATUS — Valve is in remote mode                  Bool
   //                      (1 = Remote mode, 0 = normal)
   //  status_LocalOn         STATUS — Valve is in local mode                    Bool
   //                      (1 = Local mode, 0 = normal)
   //  status_RLOff         STATUS — Valve is in ALL mode                   Bool
   //                      (1 = ALL mode, 0 = normal)
   //  ――――――――――――――――――――――――――――――――――――――――――
   // ▄▄▄▄▄▄▄▄▄▄▄▄▄▄▄▄▄▄▄▄▄▄▄▄▄▄▄▄▄▄▄▄▄▄▄▄▄▄▄▄▄▄▄▄
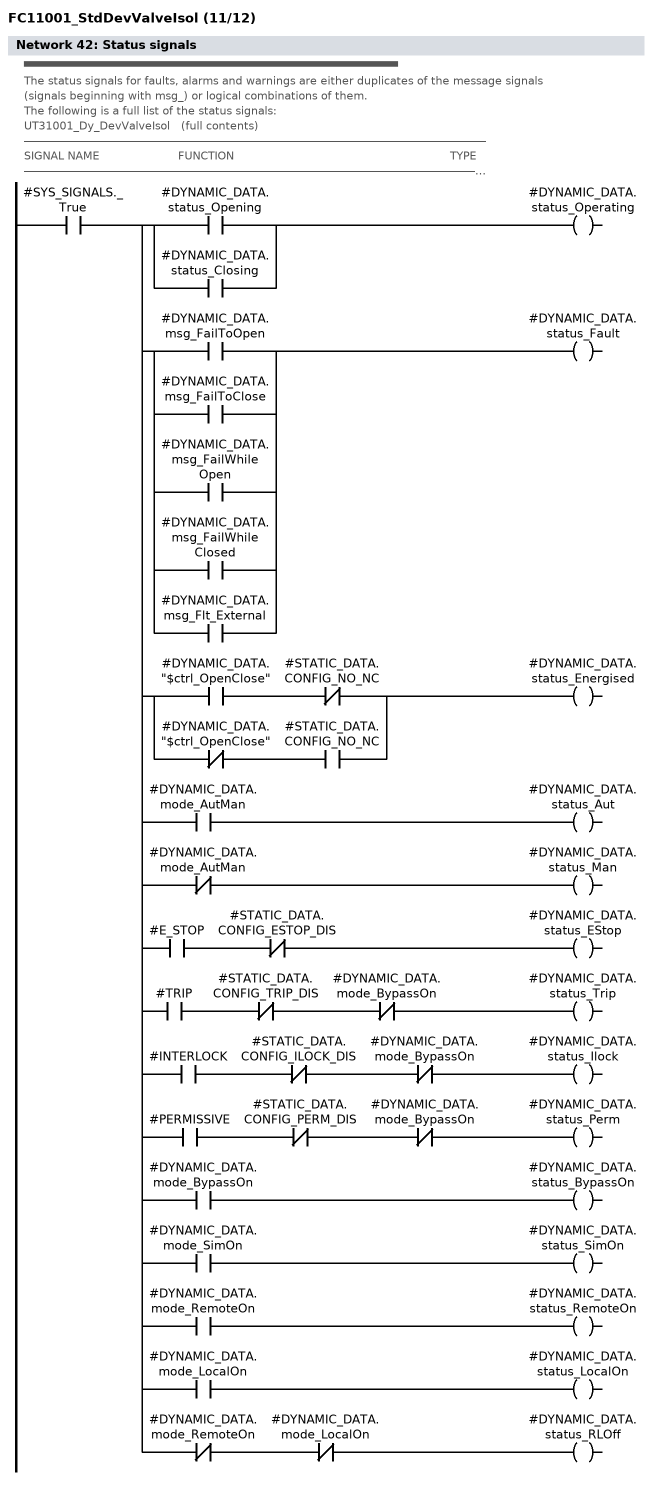
   RUNG wire#powerrail
      Contact( #SYS_SIGNALS._True )
      wire#w1
      Contact( #DYNAMIC_DATA.status_Opening )
      wire#w2
      Coil( #DYNAMIC_DATA.status_Operating )
   END_RUNG
   RUNG wire#w1
      Contact( #DYNAMIC_DATA.status_Closing )
   END_RUNG wire#w2
   RUNG wire#w1
      Contact( #DYNAMIC_DATA.msg_FailToOpen )
      wire#w3
      Coil( #DYNAMIC_DATA.status_Fault )
   END_RUNG
   RUNG wire#w1
      Contact( #DYNAMIC_DATA.msg_FailToClose )
   END_RUNG wire#w3
   RUNG wire#w1
      Contact( #DYNAMIC_DATA.msg_FailWhileOpen )
   END_RUNG wire#w3
   RUNG wire#w1
      Contact( #DYNAMIC_DATA.msg_FailWhileClosed )
   END_RUNG wire#w3
   RUNG wire#w1
      Contact( #DYNAMIC_DATA.msg_Flt_External )
   END_RUNG wire#w3
   RUNG wire#w1
      Contact( #DYNAMIC_DATA."$ctrl_OpenClose" )
      I_Contact( #STATIC_DATA.CONFIG_NO_NC )
      wire#w4
      Coil( #DYNAMIC_DATA.status_Energised )
   END_RUNG
   RUNG wire#w1
      I_Contact( #DYNAMIC_DATA."$ctrl_OpenClose" )
      Contact( #STATIC_DATA.CONFIG_NO_NC )
   END_RUNG wire#w4
   RUNG wire#w1
      Contact( #DYNAMIC_DATA.mode_AutMan )
      Coil( #DYNAMIC_DATA.status_Aut )
   END_RUNG
   RUNG wire#w1
      I_Contact( #DYNAMIC_DATA.mode_AutMan )
      Coil( #DYNAMIC_DATA.status_Man )
   END_RUNG
   RUNG wire#w1
      Contact( #E_STOP )
      I_Contact( #STATIC_DATA.CONFIG_ESTOP_DIS )
      Coil( #DYNAMIC_DATA.status_EStop )
   END_RUNG
   RUNG wire#w1
      Contact( #TRIP )
      I_Contact( #STATIC_DATA.CONFIG_TRIP_DIS )
      I_Contact( #DYNAMIC_DATA.mode_BypassOn )
      Coil( #DYNAMIC_DATA.status_Trip )
   END_RUNG
   RUNG wire#w1
      Contact( #INTERLOCK )
      I_Contact( #STATIC_DATA.CONFIG_ILOCK_DIS )
      I_Contact( #DYNAMIC_DATA.mode_BypassOn )
      Coil( #DYNAMIC_DATA.status_Ilock )
   END_RUNG
   RUNG wire#w1
      Contact( #PERMISSIVE )
      I_Contact( #STATIC_DATA.CONFIG_PERM_DIS )
      I_Contact( #DYNAMIC_DATA.mode_BypassOn )
      Coil( #DYNAMIC_DATA.status_Perm )
   END_RUNG
   RUNG wire#w1
      Contact( #DYNAMIC_DATA.mode_BypassOn )
      Coil( #DYNAMIC_DATA.status_BypassOn )
   END_RUNG
   RUNG wire#w1
      Contact( #DYNAMIC_DATA.mode_SimOn )
      Coil( #DYNAMIC_DATA.status_SimOn )
   END_RUNG
   RUNG wire#w1
      Contact( #DYNAMIC_DATA.mode_RemoteOn )
      Coil( #DYNAMIC_DATA.status_RemoteOn )
   END_RUNG
   RUNG wire#w1
      Contact( #DYNAMIC_DATA.mode_LocalOn )
      Coil( #DYNAMIC_DATA.status_LocalOn )
   END_RUNG
   RUNG wire#w1
      I_Contact( #DYNAMIC_DATA.mode_RemoteOn )
      I_Contact( #DYNAMIC_DATA.mode_LocalOn )
      Coil( #DYNAMIC_DATA.status_RLOff )
   END_RUNG
   // the same network as SCL:
   #DYNAMIC_DATA.status_Operating := #SYS_SIGNALS._True AND (#DYNAMIC_DATA.status_Opening OR #DYNAMIC_DATA.status_Closing);
   #DYNAMIC_DATA.status_Fault := #SYS_SIGNALS._True AND (#DYNAMIC_DATA.msg_FailToOpen OR #DYNAMIC_DATA.msg_FailToClose OR #DYNAMIC_DATA.msg_FailWhileOpen OR #DYNAMIC_DATA.msg_FailWhileClosed OR #DYNAMIC_DATA.msg_Flt_External);
   #DYNAMIC_DATA.status_Energised := #SYS_SIGNALS._True AND ((#DYNAMIC_DATA."$ctrl_OpenClose" AND NOT #STATIC_DATA.CONFIG_NO_NC) OR (NOT #DYNAMIC_DATA."$ctrl_OpenClose" AND #STATIC_DATA.CONFIG_NO_NC));
   #DYNAMIC_DATA.status_Aut := #SYS_SIGNALS._True AND #DYNAMIC_DATA.mode_AutMan;
   #DYNAMIC_DATA.status_Man := #SYS_SIGNALS._True AND NOT #DYNAMIC_DATA.mode_AutMan;
   #DYNAMIC_DATA.status_EStop := #SYS_SIGNALS._True AND #E_STOP AND NOT #STATIC_DATA.CONFIG_ESTOP_DIS;
   #DYNAMIC_DATA.status_Trip := #SYS_SIGNALS._True AND #TRIP AND NOT #STATIC_DATA.CONFIG_TRIP_DIS AND NOT #DYNAMIC_DATA.mode_BypassOn;
   #DYNAMIC_DATA.status_Ilock := #SYS_SIGNALS._True AND #INTERLOCK AND NOT #STATIC_DATA.CONFIG_ILOCK_DIS AND NOT #DYNAMIC_DATA.mode_BypassOn;
   #DYNAMIC_DATA.status_Perm := #SYS_SIGNALS._True AND #PERMISSIVE AND NOT #STATIC_DATA.CONFIG_PERM_DIS AND NOT #DYNAMIC_DATA.mode_BypassOn;
   #DYNAMIC_DATA.status_BypassOn := #SYS_SIGNALS._True AND #DYNAMIC_DATA.mode_BypassOn;
   #DYNAMIC_DATA.status_SimOn := #SYS_SIGNALS._True AND #DYNAMIC_DATA.mode_SimOn;
   #DYNAMIC_DATA.status_RemoteOn := #SYS_SIGNALS._True AND #DYNAMIC_DATA.mode_RemoteOn;
   #DYNAMIC_DATA.status_LocalOn := #SYS_SIGNALS._True AND #DYNAMIC_DATA.mode_LocalOn;
   #DYNAMIC_DATA.status_RLOff := #SYS_SIGNALS._True AND NOT #DYNAMIC_DATA.mode_RemoteOn AND NOT #DYNAMIC_DATA.mode_LocalOn;
END_REGION

REGION Network 43: Output driver
   // ▀▀▀▀▀▀▀▀▀▀▀▀▀▀▀▀▀▀▀▀▀▀▀▀▀▀▀▀▀▀▀▀▀▀▀▀▀▀▀▀▀▀▀▀
   // Copy the required energised/deenergised state (status_Energised) to the valve output 
   // parameter (#OPERATE)
   // ▄▄▄▄▄▄▄▄▄▄▄▄▄▄▄▄▄▄▄▄▄▄▄▄▄▄▄▄▄▄▄▄▄▄▄▄▄▄▄▄▄▄▄▄
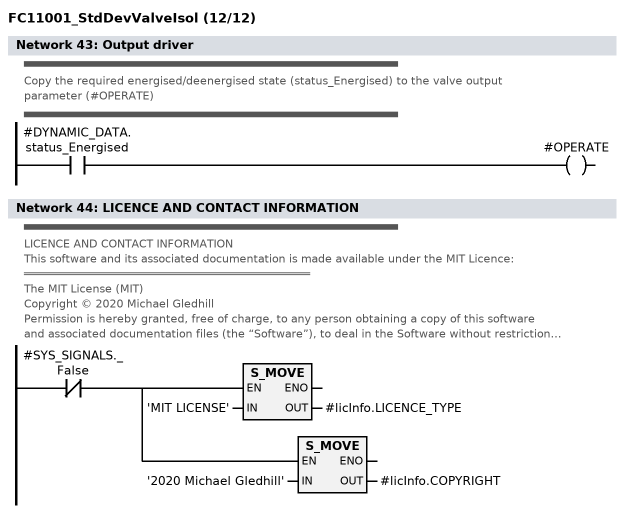
   RUNG wire#powerrail
      Contact( #DYNAMIC_DATA.status_Energised )
      Coil( #OPERATE )
   END_RUNG
   // the same network as SCL:
   #OPERATE := #DYNAMIC_DATA.status_Energised;
END_REGION

REGION Network 44: LICENCE AND CONTACT INFORMATION
   // ▀▀▀▀▀▀▀▀▀▀▀▀▀▀▀▀▀▀▀▀▀▀▀▀▀▀▀▀▀▀▀▀▀▀▀▀▀▀▀▀▀▀▀▀
   // LICENCE AND CONTACT INFORMATION
   // 
   // This software and its associated documentation is made available under the MIT Licence:
   // 
   // ════════════════════════════════════════════
   // 
   // The MIT License (MIT)
   // 
   // Copyright © 2020 Michael Gledhill
   // 
   // Permission is hereby granted, free of charge, to any person obtaining a copy of this software 
   // and associated documentation files (the “Software”), to deal in the Software without restriction, 
   // including without limitation the rights to use, copy, modify, merge, publish, distribute, 
   // sublicense, and/or sell copies of the Software, and to permit persons to whom the Software is 
   // furnished to do so, subject to the following conditions: 
   // 
   // The above copyright notice and this permission notice shall be included in all copies or 
   // substantial portions of the Software.
   // 
   // THE SOFTWARE IS PROVIDED “AS IS”, WITHOUT WARRANTY OF ANY KIND, EXPRESS OR IMPLIED, 
   // INCLUDING BUT NOT LIMITED TO THE WARRANTIES OF MERCHANTABILITY, FITNESS FOR A 
   // PARTICULAR PURPOSE AND NON-INFRINGEMENT. IN NO EVENT SHALL THE AUTHORS OR COPYRIGHT 
   // HOLDERS BE LIABLE FOR ANY CLAIM, DAMAGES OR OTHER LIABILITY, WHETHER IN AN ACTION OF 
   // CONTRACT, TORT OR OTHERWISE, ARISING FROM, OUT OF OR IN CONNECTION WITH THE SOFTWARE 
   // OR THE USE OR OTHER DEALINGS IN THE SOFTWARE.
   // 
   // ════════════════════════════════════════════
   //                    ┌────────────┐
   // You can reach the author by email here:   │  mg@practicalseries.com  │
   //                    └────────────┘
   // Questions, corrections, constructive criticism and complaints (polite ones) are invited.
   RUNG wire#powerrail
      I_Contact( #SYS_SIGNALS._False )
      wire#w1
      S_Move(in := 'MIT LICENSE', out => #licInfo.LICENCE_TYPE)
   END_RUNG
   RUNG wire#w1
      S_Move(in := '2020 Michael Gledhill', out => #licInfo.COPYRIGHT)
   END_RUNG
   // the same network as SCL:
   IF NOT #SYS_SIGNALS._False THEN
       #licInfo.LICENCE_TYPE := 'MIT LICENSE';
       #licInfo.COPYRIGHT := '2020 Michael Gledhill';
   END_IF;
END_REGION
END_FUNCTION

FUNCTION "FC11011_StdDevValve3Way" : Void   // FC11011, LAD
TITLE = Standard Module [DEVICE DRIVER] — Three-Way Valve
{ S7_Optimized_Access := 'TRUE' }
AUTHOR : M_Gledhill
FAMILY : DeviceDriver
NAME : StdDevValve3Way
VERSION : 0.8
// PRACTICAL SERIES AUTOMATION LIBRARY (PAL)   —   COPYRIGHT 2020 – M. GLEDHILL (MIT LICENCE)
//                   ———— ◆ ————
// FULL ONLINE DOCUMENTATION IS AVAILABLE AT: https://practicalseries.com/2001-pal/index.html
// stored: AutoNumber false, IsIECCheckEnabled true, SetENOAutomatically false, UDAEnableTagReadback false
   VAR_INPUT
      SYS_SIGNALS : "UT21000_Dy_SysSignals";   // Common system signals — logic and timing signals
      FBK_ENG : Bool;   // Positive energised position feedback (1 = valve energised0 = valve not energised)
      FBK_DENG : Bool;   // Positive deenergised position feedback (1 = valve deenergised 0 = valve not deenergised
      EXT_FAULT : Bool;   // Device external fault signal (1 = fault, 0 = healthy)
      E_STOP : Bool;   // Safety (E-STOP) signal (1 = ESTOP active, 0 = healthy)
      TRIP : Bool;   // Interlock (TRIP) signal (1 = TRIP active, 0 = healthy)
      INTERLOCK : Bool;   // Interlock (INTERLOCK) signal (1 = INTERLOCK active, 0 = healthy)
      PERMISSIVE : Bool;   // Interlock (PERMISSIVE) signal (1 = PERMISSIVE active, 0 = healthy)
      STATIC_DATA : "UT11011_St_DevValve3Way";   // Static data storage (UDT)
   END_VAR
   VAR_OUTPUT
      OPERATE : Bool;   // Valve operate signal (1 = energise the valve, 0 = deenergise the valve)
   END_VAR
   VAR_IN_OUT
      DYNAMIC_DATA : "UT31011_Dy_DevValve3Way";   // Dynamic data storage (UDT)
   END_VAR
   VAR_TEMP
      revInfo : "UT01000_St_SysRevision";   // Revision information for this block
      licInfo : "UT01001_St_SysLicence";   // Licensing information for this block
      calDengElapsedTime : Real;   // Calculation - Derived deenergised signal elapsed time limit
      calEngElapsedTime : Real;   // Calculation - Derived energised signal elapsed time limit
      wrkEng : Bool;   // Working - energised position feedback signal (actual or derived)
      wrkDeng : Bool;   // Working - deenergised position feedback signal (actual or derived)
      wrkCtrlPriority40 : Bool;   // Working - priority 40 condition controls the valve
      wrkCtrlPriority30 : Bool;   // Working - priority 30 condition controls the valve
      wrkCtrlPriority20 : Bool;   // Working - priority 20 condition controls the valve
      wrkCtrlPriority10 : Bool;   // Working - priority 10 condition controls the valve
      wrkCtrlPriority00 : Bool;   // Working - priority 00 condition controls the valve
      wrkCtrlAutManEngDeng : Bool;   // Working - consolidated auto/manual energise or deenergise request
      wrkTimeFbkEngSim : Real;   // Working - value of energising timer before derived energised feedback
      wrkTimeFbkDengSim : Real;   // Working - value of deenergising timer before derived deenergised feedback
      wrkInt : Int;   // Working - storage area (integer)
      wrkReal : Real;   // Working - storage area (Real)
      wrkDInt : DInt;   // Working - storage area (double integer)
   END_VAR
   VAR CONSTANT
      k_TIME_OP_MIN : Real := 0.21;   // Minimum value for the valve operation timer
   END_VAR
   VAR_TEMP   // added for the SCL form of the ladder/FBD networks
      _w1 : Bool;
      _w2 : Bool;
      _w3 : Bool;
   END_VAR
BEGIN

